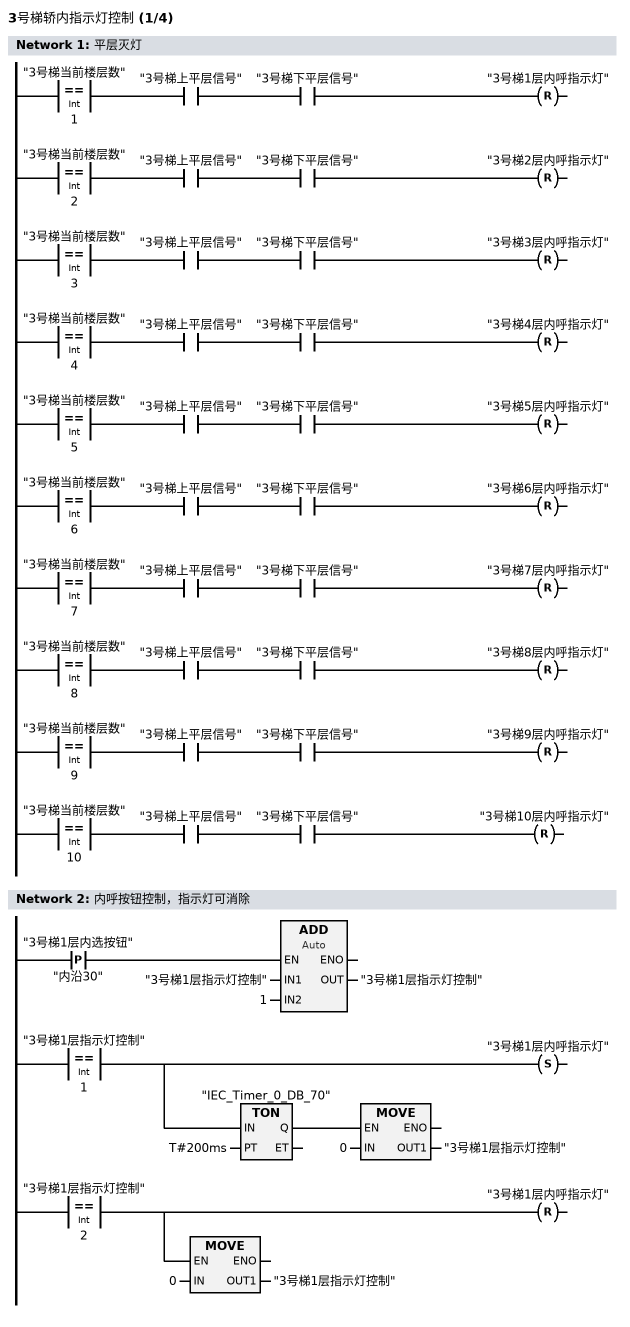
   RUNG wire#powerrail
      { S7_Templates := "SrcType := Int" } EQ_Contact(in1 := "3号梯当前楼层数", in2 := 1)
      Contact( "3号梯上平层信号" )
      Contact( "3号梯下平层信号" )
      R_Coil( "3号梯1层内呼指示灯" )
   END_RUNG
   RUNG wire#powerrail
      { S7_Templates := "SrcType := Int" } EQ_Contact(in1 := "3号梯当前楼层数", in2 := 2)
      Contact( "3号梯上平层信号" )
      Contact( "3号梯下平层信号" )
      R_Coil( "3号梯2层内呼指示灯" )
   END_RUNG
   RUNG wire#powerrail
      { S7_Templates := "SrcType := Int" } EQ_Contact(in1 := "3号梯当前楼层数", in2 := 3)
      Contact( "3号梯上平层信号" )
      Contact( "3号梯下平层信号" )
      R_Coil( "3号梯3层内呼指示灯" )
   END_RUNG
   RUNG wire#powerrail
      { S7_Templates := "SrcType := Int" } EQ_Contact(in1 := "3号梯当前楼层数", in2 := 4)
      Contact( "3号梯上平层信号" )
      Contact( "3号梯下平层信号" )
      R_Coil( "3号梯4层内呼指示灯" )
   END_RUNG
   RUNG wire#powerrail
      { S7_Templates := "SrcType := Int" } EQ_Contact(in1 := "3号梯当前楼层数", in2 := 5)
      Contact( "3号梯上平层信号" )
      Contact( "3号梯下平层信号" )
      R_Coil( "3号梯5层内呼指示灯" )
   END_RUNG
   RUNG wire#powerrail
      { S7_Templates := "SrcType := Int" } EQ_Contact(in1 := "3号梯当前楼层数", in2 := 6)
      Contact( "3号梯上平层信号" )
      Contact( "3号梯下平层信号" )
      R_Coil( "3号梯6层内呼指示灯" )
   END_RUNG
   RUNG wire#powerrail
      { S7_Templates := "SrcType := Int" } EQ_Contact(in1 := "3号梯当前楼层数", in2 := 7)
      Contact( "3号梯上平层信号" )
      Contact( "3号梯下平层信号" )
      R_Coil( "3号梯7层内呼指示灯" )
   END_RUNG
   RUNG wire#powerrail
      { S7_Templates := "SrcType := Int" } EQ_Contact(in1 := "3号梯当前楼层数", in2 := 8)
      Contact( "3号梯上平层信号" )
      Contact( "3号梯下平层信号" )
      R_Coil( "3号梯8层内呼指示灯" )
   END_RUNG
   RUNG wire#powerrail
      { S7_Templates := "SrcType := Int" } EQ_Contact(in1 := "3号梯当前楼层数", in2 := 9)
      Contact( "3号梯上平层信号" )
      Contact( "3号梯下平层信号" )
      R_Coil( "3号梯9层内呼指示灯" )
   END_RUNG
   RUNG wire#powerrail
      { S7_Templates := "SrcType := Int" } EQ_Contact(in1 := "3号梯当前楼层数", in2 := 10)
      Contact( "3号梯上平层信号" )
      Contact( "3号梯下平层信号" )
      R_Coil( "3号梯10层内呼指示灯" )
   END_RUNG
   // the same network as SCL:
   IF ("3号梯当前楼层数" = 1) AND "3号梯上平层信号" AND "3号梯下平层信号" THEN "3号梯1层内呼指示灯" := FALSE; END_IF;
   IF ("3号梯当前楼层数" = 2) AND "3号梯上平层信号" AND "3号梯下平层信号" THEN "3号梯2层内呼指示灯" := FALSE; END_IF;
   IF ("3号梯当前楼层数" = 3) AND "3号梯上平层信号" AND "3号梯下平层信号" THEN "3号梯3层内呼指示灯" := FALSE; END_IF;
   IF ("3号梯当前楼层数" = 4) AND "3号梯上平层信号" AND "3号梯下平层信号" THEN "3号梯4层内呼指示灯" := FALSE; END_IF;
   IF ("3号梯当前楼层数" = 5) AND "3号梯上平层信号" AND "3号梯下平层信号" THEN "3号梯5层内呼指示灯" := FALSE; END_IF;
   IF ("3号梯当前楼层数" = 6) AND "3号梯上平层信号" AND "3号梯下平层信号" THEN "3号梯6层内呼指示灯" := FALSE; END_IF;
   IF ("3号梯当前楼层数" = 7) AND "3号梯上平层信号" AND "3号梯下平层信号" THEN "3号梯7层内呼指示灯" := FALSE; END_IF;
   IF ("3号梯当前楼层数" = 8) AND "3号梯上平层信号" AND "3号梯下平层信号" THEN "3号梯8层内呼指示灯" := FALSE; END_IF;
   IF ("3号梯当前楼层数" = 9) AND "3号梯上平层信号" AND "3号梯下平层信号" THEN "3号梯9层内呼指示灯" := FALSE; END_IF;
   IF ("3号梯当前楼层数" = 10) AND "3号梯上平层信号" AND "3号梯下平层信号" THEN "3号梯10层内呼指示灯" := FALSE; END_IF;
END_REGION

REGION Network 2: 内呼按钮控制，指示灯可消除
   #_w1 := "3号梯1层内选按钮" AND NOT "内沿30";   // rising edge of "3号梯1层内选按钮"
   "内沿30" := "3号梯1层内选按钮";
   IF #_w1 THEN "3号梯1层指示灯控制" := "3号梯1层指示灯控制" + 1; END_IF;
   #_w2 := "3号梯1层指示灯控制" = 1;
   IF #_w2 THEN "3号梯1层内呼指示灯" := TRUE; END_IF;
   "IEC_Timer_0_DB_70".TON(IN := #_w2, PT := T#200ms);
   IF "IEC_Timer_0_DB_70".Q THEN "3号梯1层指示灯控制" := 0; END_IF;
   IF "3号梯1层指示灯控制" = 2 THEN
       "3号梯1层内呼指示灯" := FALSE;
       "3号梯1层指示灯控制" := 0;
   END_IF;
END_REGION

REGION Network 3: 内呼按钮控制，指示灯可消除
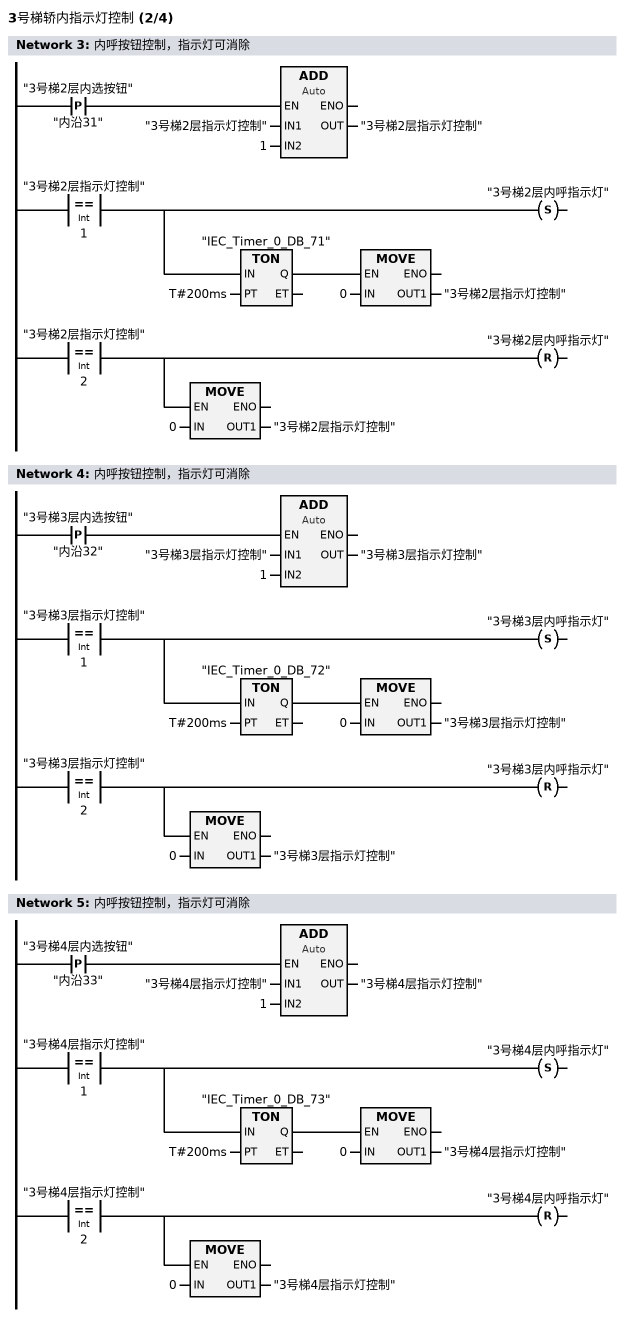
   #_w1 := "3号梯2层内选按钮" AND NOT "内沿31";   // rising edge of "3号梯2层内选按钮"
   "内沿31" := "3号梯2层内选按钮";
   IF #_w1 THEN "3号梯2层指示灯控制" := "3号梯2层指示灯控制" + 1; END_IF;
   #_w2 := "3号梯2层指示灯控制" = 1;
   IF #_w2 THEN "3号梯2层内呼指示灯" := TRUE; END_IF;
   "IEC_Timer_0_DB_71".TON(IN := #_w2, PT := T#200ms);
   IF "IEC_Timer_0_DB_71".Q THEN "3号梯2层指示灯控制" := 0; END_IF;
   IF "3号梯2层指示灯控制" = 2 THEN
       "3号梯2层内呼指示灯" := FALSE;
       "3号梯2层指示灯控制" := 0;
   END_IF;
END_REGION

REGION Network 4: 内呼按钮控制，指示灯可消除
   #_w1 := "3号梯3层内选按钮" AND NOT "内沿32";   // rising edge of "3号梯3层内选按钮"
   "内沿32" := "3号梯3层内选按钮";
   IF #_w1 THEN "3号梯3层指示灯控制" := "3号梯3层指示灯控制" + 1; END_IF;
   #_w2 := "3号梯3层指示灯控制" = 1;
   IF #_w2 THEN "3号梯3层内呼指示灯" := TRUE; END_IF;
   "IEC_Timer_0_DB_72".TON(IN := #_w2, PT := T#200ms);
   IF "IEC_Timer_0_DB_72".Q THEN "3号梯3层指示灯控制" := 0; END_IF;
   IF "3号梯3层指示灯控制" = 2 THEN
       "3号梯3层内呼指示灯" := FALSE;
       "3号梯3层指示灯控制" := 0;
   END_IF;
END_REGION

REGION Network 5: 内呼按钮控制，指示灯可消除
   #_w1 := "3号梯4层内选按钮" AND NOT "内沿33";   // rising edge of "3号梯4层内选按钮"
   "内沿33" := "3号梯4层内选按钮";
   IF #_w1 THEN "3号梯4层指示灯控制" := "3号梯4层指示灯控制" + 1; END_IF;
   #_w2 := "3号梯4层指示灯控制" = 1;
   IF #_w2 THEN "3号梯4层内呼指示灯" := TRUE; END_IF;
   "IEC_Timer_0_DB_73".TON(IN := #_w2, PT := T#200ms);
   IF "IEC_Timer_0_DB_73".Q THEN "3号梯4层指示灯控制" := 0; END_IF;
   IF "3号梯4层指示灯控制" = 2 THEN
       "3号梯4层内呼指示灯" := FALSE;
       "3号梯4层指示灯控制" := 0;
   END_IF;
END_REGION

REGION Network 6: 内呼按钮控制，指示灯可消除
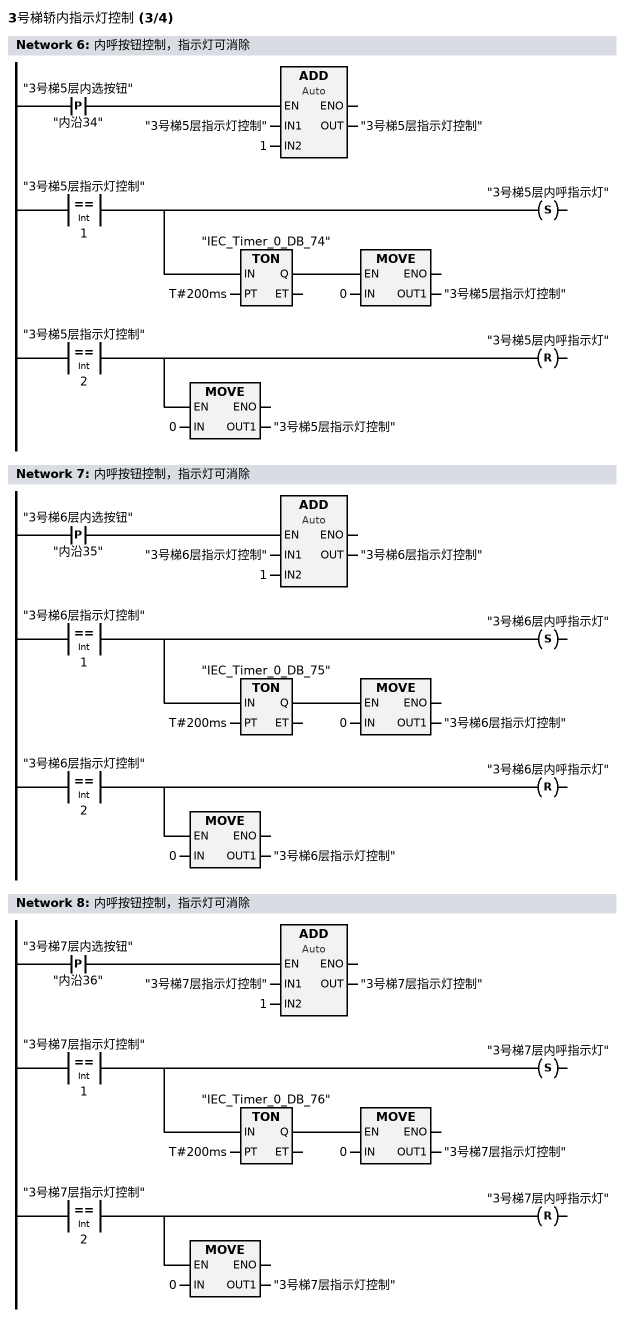
   #_w1 := "3号梯5层内选按钮" AND NOT "内沿34";   // rising edge of "3号梯5层内选按钮"
   "内沿34" := "3号梯5层内选按钮";
   IF #_w1 THEN "3号梯5层指示灯控制" := "3号梯5层指示灯控制" + 1; END_IF;
   #_w2 := "3号梯5层指示灯控制" = 1;
   IF #_w2 THEN "3号梯5层内呼指示灯" := TRUE; END_IF;
   "IEC_Timer_0_DB_74".TON(IN := #_w2, PT := T#200ms);
   IF "IEC_Timer_0_DB_74".Q THEN "3号梯5层指示灯控制" := 0; END_IF;
   IF "3号梯5层指示灯控制" = 2 THEN
       "3号梯5层内呼指示灯" := FALSE;
       "3号梯5层指示灯控制" := 0;
   END_IF;
END_REGION

REGION Network 7: 内呼按钮控制，指示灯可消除
   #_w1 := "3号梯6层内选按钮" AND NOT "内沿35";   // rising edge of "3号梯6层内选按钮"
   "内沿35" := "3号梯6层内选按钮";
   IF #_w1 THEN "3号梯6层指示灯控制" := "3号梯6层指示灯控制" + 1; END_IF;
   #_w2 := "3号梯6层指示灯控制" = 1;
   IF #_w2 THEN "3号梯6层内呼指示灯" := TRUE; END_IF;
   "IEC_Timer_0_DB_75".TON(IN := #_w2, PT := T#200ms);
   IF "IEC_Timer_0_DB_75".Q THEN "3号梯6层指示灯控制" := 0; END_IF;
   IF "3号梯6层指示灯控制" = 2 THEN
       "3号梯6层内呼指示灯" := FALSE;
       "3号梯6层指示灯控制" := 0;
   END_IF;
END_REGION

REGION Network 8: 内呼按钮控制，指示灯可消除
   #_w1 := "3号梯7层内选按钮" AND NOT "内沿36";   // rising edge of "3号梯7层内选按钮"
   "内沿36" := "3号梯7层内选按钮";
   IF #_w1 THEN "3号梯7层指示灯控制" := "3号梯7层指示灯控制" + 1; END_IF;
   #_w2 := "3号梯7层指示灯控制" = 1;
   IF #_w2 THEN "3号梯7层内呼指示灯" := TRUE; END_IF;
   "IEC_Timer_0_DB_76".TON(IN := #_w2, PT := T#200ms);
   IF "IEC_Timer_0_DB_76".Q THEN "3号梯7层指示灯控制" := 0; END_IF;
   IF "3号梯7层指示灯控制" = 2 THEN
       "3号梯7层内呼指示灯" := FALSE;
       "3号梯7层指示灯控制" := 0;
   END_IF;
END_REGION

REGION Network 9: 内呼按钮控制，指示灯可消除
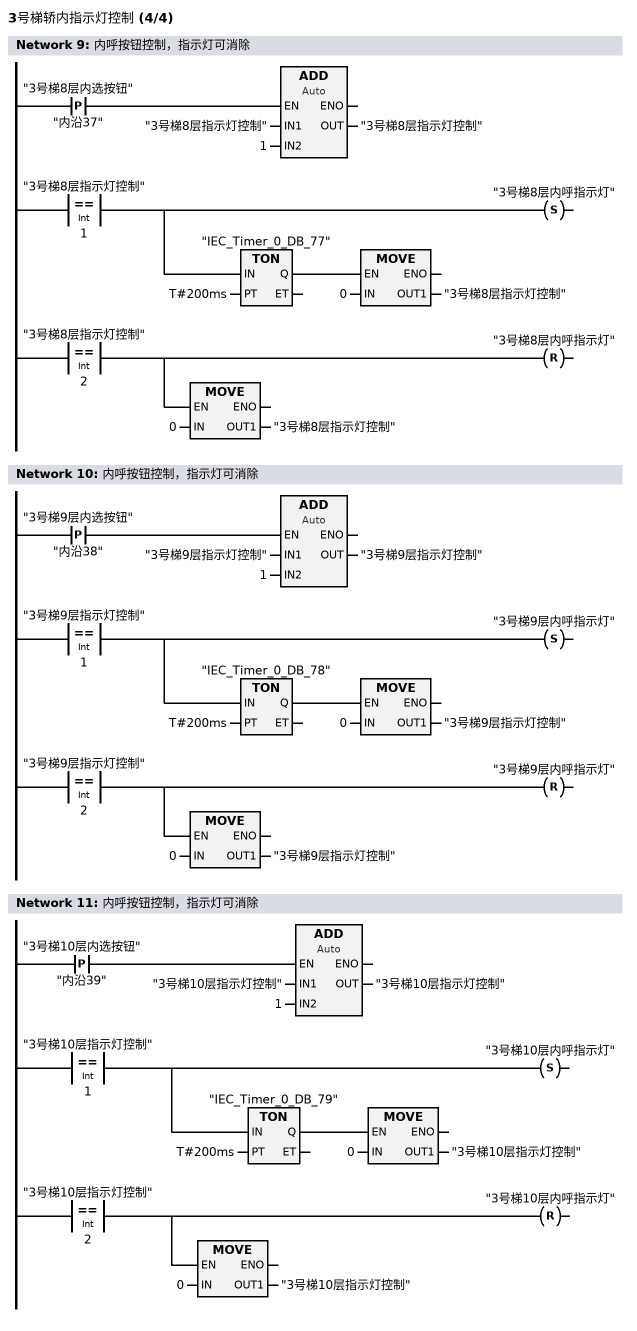
   #_w1 := "3号梯8层内选按钮" AND NOT "内沿37";   // rising edge of "3号梯8层内选按钮"
   "内沿37" := "3号梯8层内选按钮";
   IF #_w1 THEN "3号梯8层指示灯控制" := "3号梯8层指示灯控制" + 1; END_IF;
   #_w2 := "3号梯8层指示灯控制" = 1;
   IF #_w2 THEN "3号梯8层内呼指示灯" := TRUE; END_IF;
   "IEC_Timer_0_DB_77".TON(IN := #_w2, PT := T#200ms);
   IF "IEC_Timer_0_DB_77".Q THEN "3号梯8层指示灯控制" := 0; END_IF;
   IF "3号梯8层指示灯控制" = 2 THEN
       "3号梯8层内呼指示灯" := FALSE;
       "3号梯8层指示灯控制" := 0;
   END_IF;
END_REGION

REGION Network 10: 内呼按钮控制，指示灯可消除
   #_w1 := "3号梯9层内选按钮" AND NOT "内沿38";   // rising edge of "3号梯9层内选按钮"
   "内沿38" := "3号梯9层内选按钮";
   IF #_w1 THEN "3号梯9层指示灯控制" := "3号梯9层指示灯控制" + 1; END_IF;
   #_w2 := "3号梯9层指示灯控制" = 1;
   IF #_w2 THEN "3号梯9层内呼指示灯" := TRUE; END_IF;
   "IEC_Timer_0_DB_78".TON(IN := #_w2, PT := T#200ms);
   IF "IEC_Timer_0_DB_78".Q THEN "3号梯9层指示灯控制" := 0; END_IF;
   IF "3号梯9层指示灯控制" = 2 THEN
       "3号梯9层内呼指示灯" := FALSE;
       "3号梯9层指示灯控制" := 0;
   END_IF;
END_REGION

REGION Network 11: 内呼按钮控制，指示灯可消除
   #_w1 := "3号梯10层内选按钮" AND NOT "内沿39";   // rising edge of "3号梯10层内选按钮"
   "内沿39" := "3号梯10层内选按钮";
   IF #_w1 THEN "3号梯10层指示灯控制" := "3号梯10层指示灯控制" + 1; END_IF;
   #_w2 := "3号梯10层指示灯控制" = 1;
   IF #_w2 THEN "3号梯10层内呼指示灯" := TRUE; END_IF;
   "IEC_Timer_0_DB_79".TON(IN := #_w2, PT := T#200ms);
   IF "IEC_Timer_0_DB_79".Q THEN "3号梯10层指示灯控制" := 0; END_IF;
   IF "3号梯10层指示灯控制" = 2 THEN
       "3号梯10层内呼指示灯" := FALSE;
       "3号梯10层指示灯控制" := 0;
   END_IF;
END_REGION
END_FUNCTION

FUNCTION "3号梯保护程序" : Void   // FC41, LAD
{ S7_Optimized_Access := 'TRUE' }
VERSION : 0.1
BEGIN

REGION Network 1: 休眠管理
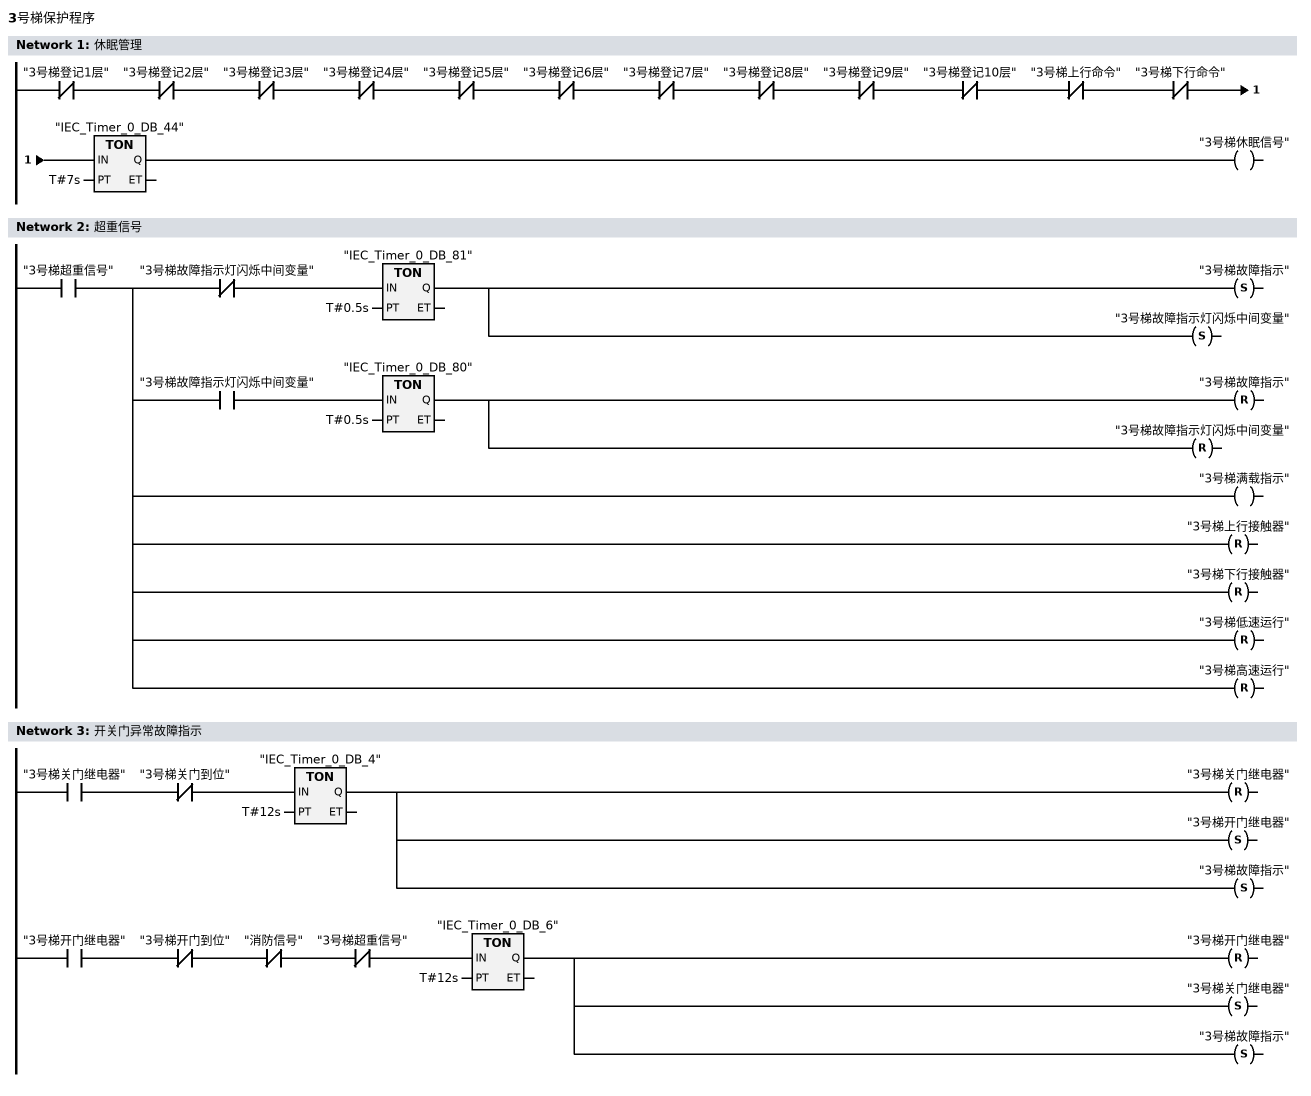
   "IEC_Timer_0_DB_44".TON(IN := NOT "3号梯登记1层" AND NOT "3号梯登记2层" AND NOT "3号梯登记3层" AND NOT "3号梯登记4层" AND NOT "3号梯登记5层" AND NOT "3号梯登记6层" AND NOT "3号梯登记7层" AND NOT "3号梯登记8层" AND NOT "3号梯登记9层" AND NOT "3号梯登记10层" AND NOT "3号梯上行命令" AND NOT "3号梯下行命令",
                           PT := T#7s);
   "3号梯休眠信号" := "IEC_Timer_0_DB_44".Q;
END_REGION

REGION Network 2: 超重信号
   "IEC_Timer_0_DB_81".TON(IN := "3号梯超重信号" AND NOT "3号梯故障指示灯闪烁中间变量", PT := T#0.5s);
   IF "IEC_Timer_0_DB_81".Q THEN
       "3号梯故障指示" := TRUE;
       "3号梯故障指示灯闪烁中间变量" := TRUE;
   END_IF;
   "IEC_Timer_0_DB_80".TON(IN := "3号梯超重信号" AND "3号梯故障指示灯闪烁中间变量", PT := T#0.5s);
   IF "IEC_Timer_0_DB_80".Q THEN
       "3号梯故障指示" := FALSE;
       "3号梯故障指示灯闪烁中间变量" := FALSE;
   END_IF;
   "3号梯满载指示" := "3号梯超重信号";
   IF "3号梯超重信号" THEN
       "3号梯上行接触器" := FALSE;
       "3号梯下行接触器" := FALSE;
       "3号梯低速运行" := FALSE;
       "3号梯高速运行" := FALSE;
   END_IF;
END_REGION

REGION Network 3: 开关门异常故障指示
   "IEC_Timer_0_DB_4".TON(IN := "3号梯关门继电器" AND NOT "3号梯关门到位", PT := T#12s);
   IF "IEC_Timer_0_DB_4".Q THEN
       "3号梯关门继电器" := FALSE;
       "3号梯开门继电器" := TRUE;
       "3号梯故障指示" := TRUE;
   END_IF;
   "IEC_Timer_0_DB_6".TON(IN := "3号梯开门继电器" AND NOT "3号梯开门到位" AND NOT "消防信号" AND NOT "3号梯超重信号", PT := T#12s);
   IF "IEC_Timer_0_DB_6".Q THEN
       "3号梯开门继电器" := FALSE;
       "3号梯关门继电器" := TRUE;
       "3号梯故障指示" := TRUE;
   END_IF;
END_REGION
END_FUNCTION

FUNCTION "2号梯保护程序" : Void   // FC42, LAD
{ S7_Optimized_Access := 'TRUE' }
VERSION : 0.1
BEGIN

REGION Network 1: 休眠管理
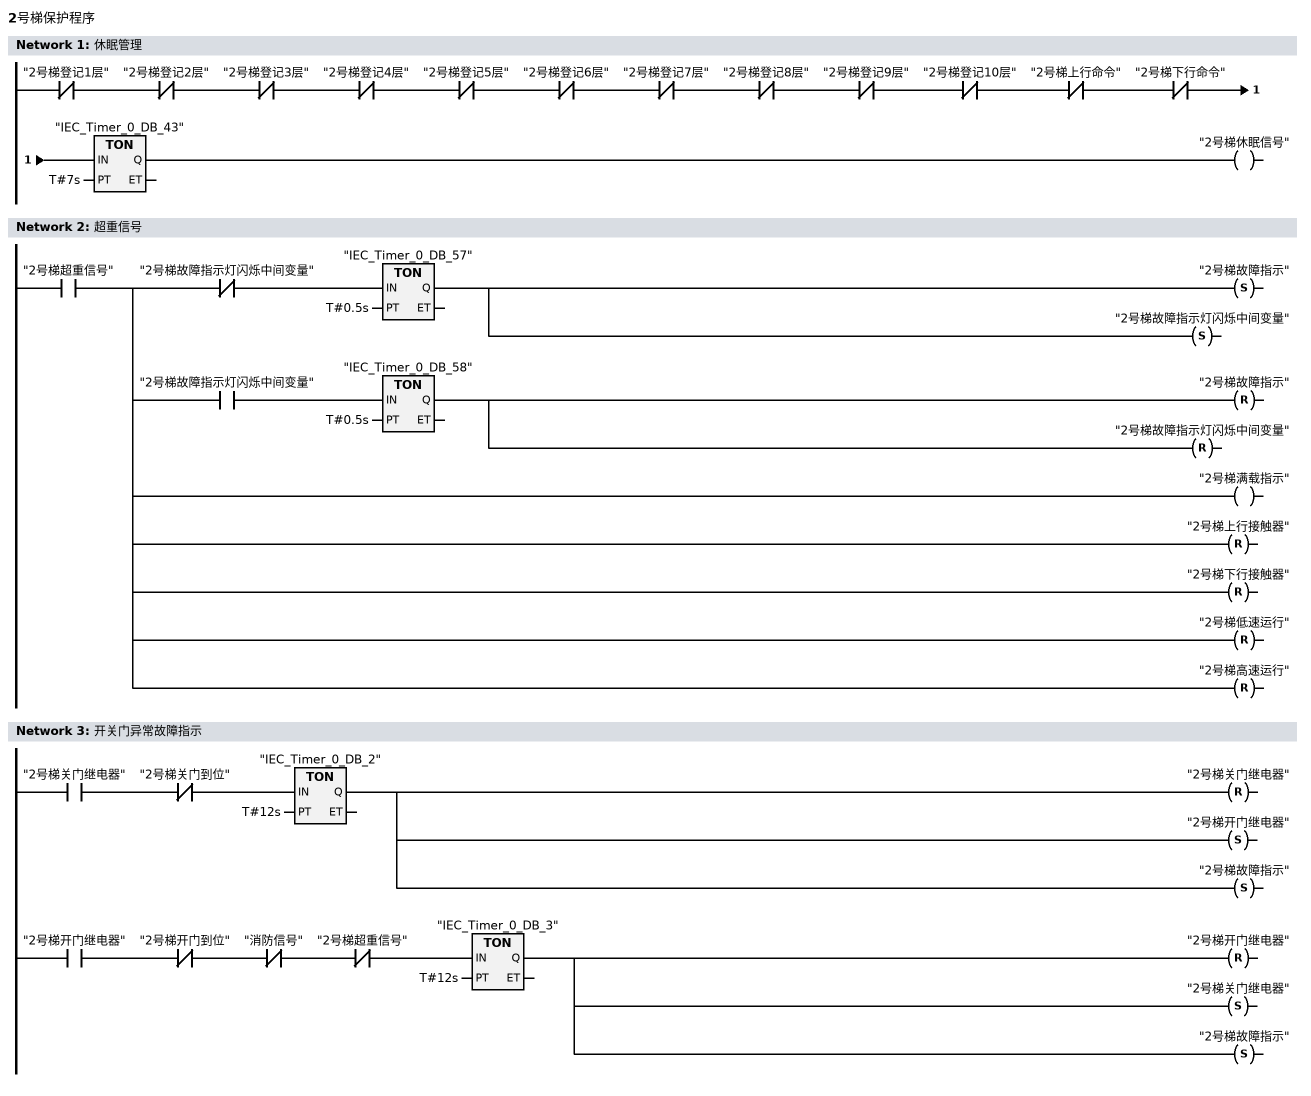
   "IEC_Timer_0_DB_43".TON(IN := NOT "2号梯登记1层" AND NOT "2号梯登记2层" AND NOT "2号梯登记3层" AND NOT "2号梯登记4层" AND NOT "2号梯登记5层" AND NOT "2号梯登记6层" AND NOT "2号梯登记7层" AND NOT "2号梯登记8层" AND NOT "2号梯登记9层" AND NOT "2号梯登记10层" AND NOT "2号梯上行命令" AND NOT "2号梯下行命令",
                           PT := T#7s);
   "2号梯休眠信号" := "IEC_Timer_0_DB_43".Q;
END_REGION

REGION Network 2: 超重信号
   "IEC_Timer_0_DB_57".TON(IN := "2号梯超重信号" AND NOT "2号梯故障指示灯闪烁中间变量", PT := T#0.5s);
   IF "IEC_Timer_0_DB_57".Q THEN
       "2号梯故障指示" := TRUE;
       "2号梯故障指示灯闪烁中间变量" := TRUE;
   END_IF;
   "IEC_Timer_0_DB_58".TON(IN := "2号梯超重信号" AND "2号梯故障指示灯闪烁中间变量", PT := T#0.5s);
   IF "IEC_Timer_0_DB_58".Q THEN
       "2号梯故障指示" := FALSE;
       "2号梯故障指示灯闪烁中间变量" := FALSE;
   END_IF;
   "2号梯满载指示" := "2号梯超重信号";
   IF "2号梯超重信号" THEN
       "2号梯上行接触器" := FALSE;
       "2号梯下行接触器" := FALSE;
       "2号梯低速运行" := FALSE;
       "2号梯高速运行" := FALSE;
   END_IF;
END_REGION

REGION Network 3: 开关门异常故障指示
   "IEC_Timer_0_DB_2".TON(IN := "2号梯关门继电器" AND NOT "2号梯关门到位", PT := T#12s);
   IF "IEC_Timer_0_DB_2".Q THEN
       "2号梯关门继电器" := FALSE;
       "2号梯开门继电器" := TRUE;
       "2号梯故障指示" := TRUE;
   END_IF;
   "IEC_Timer_0_DB_3".TON(IN := "2号梯开门继电器" AND NOT "2号梯开门到位" AND NOT "消防信号" AND NOT "2号梯超重信号", PT := T#12s);
   IF "IEC_Timer_0_DB_3".Q THEN
       "2号梯开门继电器" := FALSE;
       "2号梯关门继电器" := TRUE;
       "2号梯故障指示" := TRUE;
   END_IF;
END_REGION
END_FUNCTION

FUNCTION "3号梯错误指令消除" : Void   // FC43, LAD
{ S7_Optimized_Access := 'TRUE' }
VERSION : 0.1
BEGIN

REGION Network 1: 最上端/最下端时， 消除内呼信号
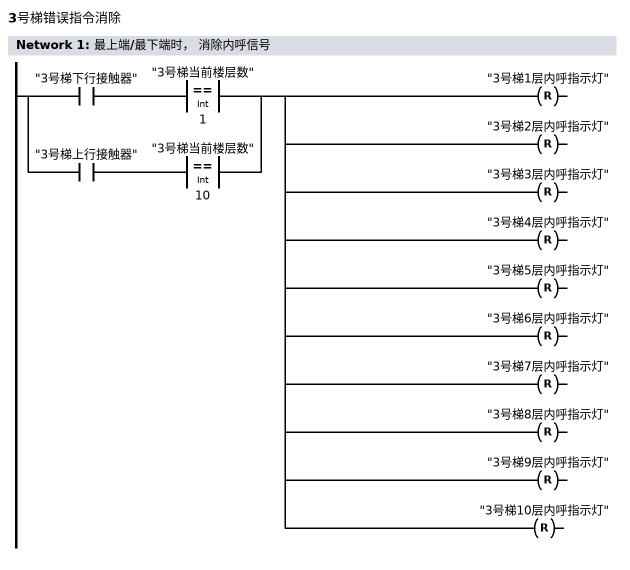
   RUNG wire#powerrail
      Contact( "3号梯下行接触器" )
      { S7_Templates := "SrcType := Int" } EQ_Contact(in1 := "3号梯当前楼层数", in2 := 1)
      wire#w1
      R_Coil( "3号梯1层内呼指示灯" )
   END_RUNG
   RUNG wire#powerrail
      Contact( "3号梯上行接触器" )
      { S7_Templates := "SrcType := Int" } EQ_Contact(in1 := "3号梯当前楼层数", in2 := 10)
   END_RUNG wire#w1
   RUNG wire#w1
      R_Coil( "3号梯2层内呼指示灯" )
   END_RUNG
   RUNG wire#w1
      R_Coil( "3号梯3层内呼指示灯" )
   END_RUNG
   RUNG wire#w1
      R_Coil( "3号梯4层内呼指示灯" )
   END_RUNG
   RUNG wire#w1
      R_Coil( "3号梯5层内呼指示灯" )
   END_RUNG
   RUNG wire#w1
      R_Coil( "3号梯6层内呼指示灯" )
   END_RUNG
   RUNG wire#w1
      R_Coil( "3号梯7层内呼指示灯" )
   END_RUNG
   RUNG wire#w1
      R_Coil( "3号梯8层内呼指示灯" )
   END_RUNG
   RUNG wire#w1
      R_Coil( "3号梯9层内呼指示灯" )
   END_RUNG
   RUNG wire#w1
      R_Coil( "3号梯10层内呼指示灯" )
   END_RUNG
   // the same network as SCL:
   IF ("3号梯下行接触器" AND ("3号梯当前楼层数" = 1)) OR ("3号梯上行接触器" AND ("3号梯当前楼层数" = 10)) THEN
       "3号梯1层内呼指示灯" := FALSE;
       "3号梯2层内呼指示灯" := FALSE;
       "3号梯3层内呼指示灯" := FALSE;
       "3号梯4层内呼指示灯" := FALSE;
       "3号梯5层内呼指示灯" := FALSE;
       "3号梯6层内呼指示灯" := FALSE;
       "3号梯7层内呼指示灯" := FALSE;
       "3号梯8层内呼指示灯" := FALSE;
       "3号梯9层内呼指示灯" := FALSE;
       "3号梯10层内呼指示灯" := FALSE;
   END_IF;
END_REGION
END_FUNCTION

FUNCTION "2号梯错误指令消除" : Void   // FC44, LAD
{ S7_Optimized_Access := 'TRUE' }
VERSION : 0.1
BEGIN

REGION Network 1: 最上端/最下端时， 消除内呼信号
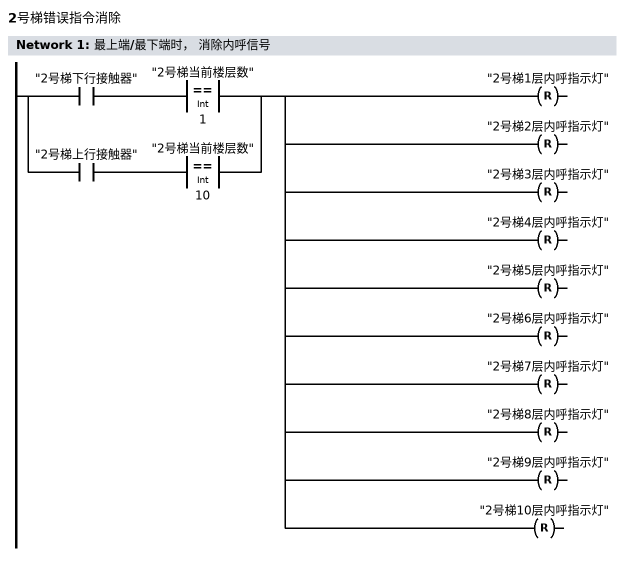
   RUNG wire#powerrail
      Contact( "2号梯下行接触器" )
      { S7_Templates := "SrcType := Int" } EQ_Contact(in1 := "2号梯当前楼层数", in2 := 1)
      wire#w1
      R_Coil( "2号梯1层内呼指示灯" )
   END_RUNG
   RUNG wire#powerrail
      Contact( "2号梯上行接触器" )
      { S7_Templates := "SrcType := Int" } EQ_Contact(in1 := "2号梯当前楼层数", in2 := 10)
   END_RUNG wire#w1
   RUNG wire#w1
      R_Coil( "2号梯2层内呼指示灯" )
   END_RUNG
   RUNG wire#w1
      R_Coil( "2号梯3层内呼指示灯" )
   END_RUNG
   RUNG wire#w1
      R_Coil( "2号梯4层内呼指示灯" )
   END_RUNG
   RUNG wire#w1
      R_Coil( "2号梯5层内呼指示灯" )
   END_RUNG
   RUNG wire#w1
      R_Coil( "2号梯6层内呼指示灯" )
   END_RUNG
   RUNG wire#w1
      R_Coil( "2号梯7层内呼指示灯" )
   END_RUNG
   RUNG wire#w1
      R_Coil( "2号梯8层内呼指示灯" )
   END_RUNG
   RUNG wire#w1
      R_Coil( "2号梯9层内呼指示灯" )
   END_RUNG
   RUNG wire#w1
      R_Coil( "2号梯10层内呼指示灯" )
   END_RUNG
   // the same network as SCL:
   IF ("2号梯下行接触器" AND ("2号梯当前楼层数" = 1)) OR ("2号梯上行接触器" AND ("2号梯当前楼层数" = 10)) THEN
       "2号梯1层内呼指示灯" := FALSE;
       "2号梯2层内呼指示灯" := FALSE;
       "2号梯3层内呼指示灯" := FALSE;
       "2号梯4层内呼指示灯" := FALSE;
       "2号梯5层内呼指示灯" := FALSE;
       "2号梯6层内呼指示灯" := FALSE;
       "2号梯7层内呼指示灯" := FALSE;
       "2号梯8层内呼指示灯" := FALSE;
       "2号梯9层内呼指示灯" := FALSE;
       "2号梯10层内呼指示灯" := FALSE;
   END_IF;
END_REGION
END_FUNCTION

FUNCTION "2号梯检修" : Void   // FC45, LAD
{ S7_Optimized_Access := 'TRUE' }
VERSION : 0.1
   VAR_TEMP   // added for the SCL form of the ladder/FBD networks
      _w1 : Bool;
   END_VAR
BEGIN

REGION Network 1: 检修
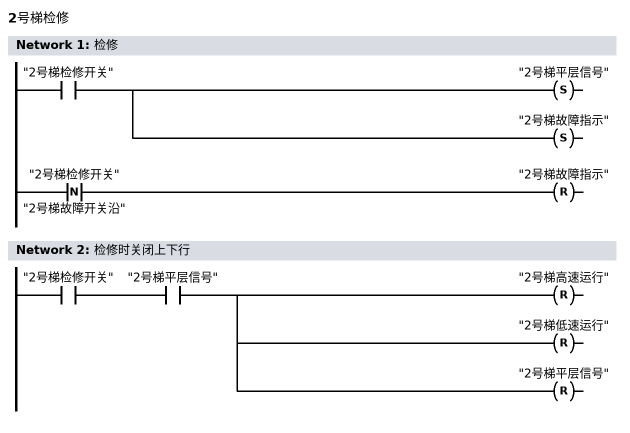
   RUNG wire#powerrail
      Contact( "2号梯检修开关" )
      wire#w1
      S_Coil( "2号梯平层信号" )
   END_RUNG
   RUNG wire#w1
      S_Coil( "2号梯故障指示" )
   END_RUNG
   RUNG wire#powerrail
      N_Contact(operand := "2号梯检修开关", bit := "2号梯故障开关沿")
      R_Coil( "2号梯故障指示" )
   END_RUNG
   // the same network as SCL:
   IF "2号梯检修开关" THEN
       "2号梯平层信号" := TRUE;
       "2号梯故障指示" := TRUE;
   END_IF;
   #_w1 := NOT "2号梯检修开关" AND "2号梯故障开关沿";   // falling edge of "2号梯检修开关"
   "2号梯故障开关沿" := "2号梯检修开关";
   IF #_w1 THEN "2号梯故障指示" := FALSE; END_IF;
END_REGION

REGION Network 2: 检修时关闭上下行
   RUNG wire#powerrail
      Contact( "2号梯检修开关" )
      Contact( "2号梯平层信号" )
      wire#w1
      R_Coil( "2号梯高速运行" )
   END_RUNG
   RUNG wire#w1
      R_Coil( "2号梯低速运行" )
   END_RUNG
   RUNG wire#w1
      R_Coil( "2号梯平层信号" )
   END_RUNG
   // the same network as SCL:
   IF "2号梯检修开关" AND "2号梯平层信号" THEN
       "2号梯高速运行" := FALSE;
       "2号梯低速运行" := FALSE;
       "2号梯平层信号" := FALSE;
   END_IF;
END_REGION
END_FUNCTION

FUNCTION "3号梯检修" : Void   // FC46, LAD
{ S7_Optimized_Access := 'TRUE' }
VERSION : 0.1
   VAR_TEMP   // added for the SCL form of the ladder/FBD networks
      _w1 : Bool;
   END_VAR
BEGIN

REGION Network 1: 检修
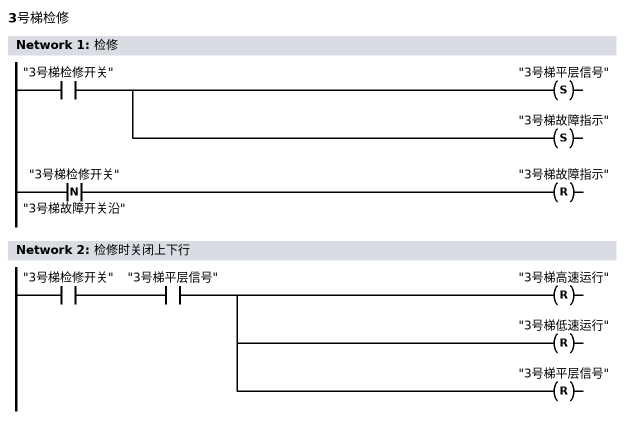
   RUNG wire#powerrail
      Contact( "3号梯检修开关" )
      wire#w1
      S_Coil( "3号梯平层信号" )
   END_RUNG
   RUNG wire#w1
      S_Coil( "3号梯故障指示" )
   END_RUNG
   RUNG wire#powerrail
      N_Contact(operand := "3号梯检修开关", bit := "3号梯故障开关沿")
      R_Coil( "3号梯故障指示" )
   END_RUNG
   // the same network as SCL:
   IF "3号梯检修开关" THEN
       "3号梯平层信号" := TRUE;
       "3号梯故障指示" := TRUE;
   END_IF;
   #_w1 := NOT "3号梯检修开关" AND "3号梯故障开关沿";   // falling edge of "3号梯检修开关"
   "3号梯故障开关沿" := "3号梯检修开关";
   IF #_w1 THEN "3号梯故障指示" := FALSE; END_IF;
END_REGION

REGION Network 2: 检修时关闭上下行
   RUNG wire#powerrail
      Contact( "3号梯检修开关" )
      Contact( "3号梯平层信号" )
      wire#w1
      R_Coil( "3号梯高速运行" )
   END_RUNG
   RUNG wire#w1
      R_Coil( "3号梯低速运行" )
   END_RUNG
   RUNG wire#w1
      R_Coil( "3号梯平层信号" )
   END_RUNG
   // the same network as SCL:
   IF "3号梯检修开关" AND "3号梯平层信号" THEN
       "3号梯高速运行" := FALSE;
       "3号梯低速运行" := FALSE;
       "3号梯平层信号" := FALSE;
   END_IF;
END_REGION
END_FUNCTION

FUNCTION "io_output" : Void   // FC47, LAD
{ S7_Optimized_Access := 'TRUE' }
VERSION : 0.1
BEGIN

REGION Network 1: 1号梯外呼上行绑定
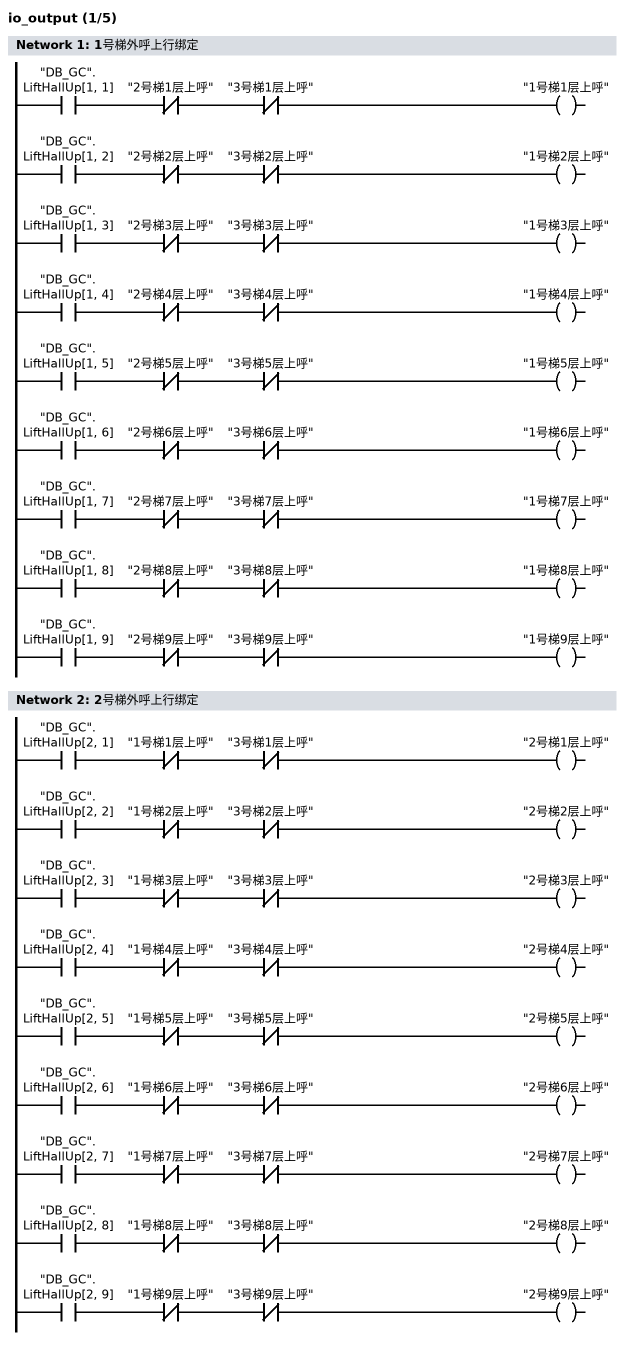
   RUNG wire#powerrail
      Contact( "DB_GC".LiftHallUp[1, 1] )
      I_Contact( "2号梯1层上呼" )
      I_Contact( "3号梯1层上呼" )
      Coil( "1号梯1层上呼" )
   END_RUNG
   RUNG wire#powerrail
      Contact( "DB_GC".LiftHallUp[1, 2] )
      I_Contact( "2号梯2层上呼" )
      I_Contact( "3号梯2层上呼" )
      Coil( "1号梯2层上呼" )
   END_RUNG
   RUNG wire#powerrail
      Contact( "DB_GC".LiftHallUp[1, 3] )
      I_Contact( "2号梯3层上呼" )
      I_Contact( "3号梯3层上呼" )
      Coil( "1号梯3层上呼" )
   END_RUNG
   RUNG wire#powerrail
      Contact( "DB_GC".LiftHallUp[1, 4] )
      I_Contact( "2号梯4层上呼" )
      I_Contact( "3号梯4层上呼" )
      Coil( "1号梯4层上呼" )
   END_RUNG
   RUNG wire#powerrail
      Contact( "DB_GC".LiftHallUp[1, 5] )
      I_Contact( "2号梯5层上呼" )
      I_Contact( "3号梯5层上呼" )
      Coil( "1号梯5层上呼" )
   END_RUNG
   RUNG wire#powerrail
      Contact( "DB_GC".LiftHallUp[1, 6] )
      I_Contact( "2号梯6层上呼" )
      I_Contact( "3号梯6层上呼" )
      Coil( "1号梯6层上呼" )
   END_RUNG
   RUNG wire#powerrail
      Contact( "DB_GC".LiftHallUp[1, 7] )
      I_Contact( "2号梯7层上呼" )
      I_Contact( "3号梯7层上呼" )
      Coil( "1号梯7层上呼" )
   END_RUNG
   RUNG wire#powerrail
      Contact( "DB_GC".LiftHallUp[1, 8] )
      I_Contact( "2号梯8层上呼" )
      I_Contact( "3号梯8层上呼" )
      Coil( "1号梯8层上呼" )
   END_RUNG
   RUNG wire#powerrail
      Contact( "DB_GC".LiftHallUp[1, 9] )
      I_Contact( "2号梯9层上呼" )
      I_Contact( "3号梯9层上呼" )
      Coil( "1号梯9层上呼" )
   END_RUNG
   // the same network as SCL:
   "1号梯1层上呼" := "DB_GC".LiftHallUp[1, 1] AND NOT "2号梯1层上呼" AND NOT "3号梯1层上呼";
   "1号梯2层上呼" := "DB_GC".LiftHallUp[1, 2] AND NOT "2号梯2层上呼" AND NOT "3号梯2层上呼";
   "1号梯3层上呼" := "DB_GC".LiftHallUp[1, 3] AND NOT "2号梯3层上呼" AND NOT "3号梯3层上呼";
   "1号梯4层上呼" := "DB_GC".LiftHallUp[1, 4] AND NOT "2号梯4层上呼" AND NOT "3号梯4层上呼";
   "1号梯5层上呼" := "DB_GC".LiftHallUp[1, 5] AND NOT "2号梯5层上呼" AND NOT "3号梯5层上呼";
   "1号梯6层上呼" := "DB_GC".LiftHallUp[1, 6] AND NOT "2号梯6层上呼" AND NOT "3号梯6层上呼";
   "1号梯7层上呼" := "DB_GC".LiftHallUp[1, 7] AND NOT "2号梯7层上呼" AND NOT "3号梯7层上呼";
   "1号梯8层上呼" := "DB_GC".LiftHallUp[1, 8] AND NOT "2号梯8层上呼" AND NOT "3号梯8层上呼";
   "1号梯9层上呼" := "DB_GC".LiftHallUp[1, 9] AND NOT "2号梯9层上呼" AND NOT "3号梯9层上呼";
END_REGION

REGION Network 2: 2号梯外呼上行绑定
   RUNG wire#powerrail
      Contact( "DB_GC".LiftHallUp[2, 1] )
      I_Contact( "1号梯1层上呼" )
      I_Contact( "3号梯1层上呼" )
      Coil( "2号梯1层上呼" )
   END_RUNG
   RUNG wire#powerrail
      Contact( "DB_GC".LiftHallUp[2, 2] )
      I_Contact( "1号梯2层上呼" )
      I_Contact( "3号梯2层上呼" )
      Coil( "2号梯2层上呼" )
   END_RUNG
   RUNG wire#powerrail
      Contact( "DB_GC".LiftHallUp[2, 3] )
      I_Contact( "1号梯3层上呼" )
      I_Contact( "3号梯3层上呼" )
      Coil( "2号梯3层上呼" )
   END_RUNG
   RUNG wire#powerrail
      Contact( "DB_GC".LiftHallUp[2, 4] )
      I_Contact( "1号梯4层上呼" )
      I_Contact( "3号梯4层上呼" )
      Coil( "2号梯4层上呼" )
   END_RUNG
   RUNG wire#powerrail
      Contact( "DB_GC".LiftHallUp[2, 5] )
      I_Contact( "1号梯5层上呼" )
      I_Contact( "3号梯5层上呼" )
      Coil( "2号梯5层上呼" )
   END_RUNG
   RUNG wire#powerrail
      Contact( "DB_GC".LiftHallUp[2, 6] )
      I_Contact( "1号梯6层上呼" )
      I_Contact( "3号梯6层上呼" )
      Coil( "2号梯6层上呼" )
   END_RUNG
   RUNG wire#powerrail
      Contact( "DB_GC".LiftHallUp[2, 7] )
      I_Contact( "1号梯7层上呼" )
      I_Contact( "3号梯7层上呼" )
      Coil( "2号梯7层上呼" )
   END_RUNG
   RUNG wire#powerrail
      Contact( "DB_GC".LiftHallUp[2, 8] )
      I_Contact( "1号梯8层上呼" )
      I_Contact( "3号梯8层上呼" )
      Coil( "2号梯8层上呼" )
   END_RUNG
   RUNG wire#powerrail
      Contact( "DB_GC".LiftHallUp[2, 9] )
      I_Contact( "1号梯9层上呼" )
      I_Contact( "3号梯9层上呼" )
      Coil( "2号梯9层上呼" )
   END_RUNG
   // the same network as SCL:
   "2号梯1层上呼" := "DB_GC".LiftHallUp[2, 1] AND NOT "1号梯1层上呼" AND NOT "3号梯1层上呼";
   "2号梯2层上呼" := "DB_GC".LiftHallUp[2, 2] AND NOT "1号梯2层上呼" AND NOT "3号梯2层上呼";
   "2号梯3层上呼" := "DB_GC".LiftHallUp[2, 3] AND NOT "1号梯3层上呼" AND NOT "3号梯3层上呼";
   "2号梯4层上呼" := "DB_GC".LiftHallUp[2, 4] AND NOT "1号梯4层上呼" AND NOT "3号梯4层上呼";
   "2号梯5层上呼" := "DB_GC".LiftHallUp[2, 5] AND NOT "1号梯5层上呼" AND NOT "3号梯5层上呼";
   "2号梯6层上呼" := "DB_GC".LiftHallUp[2, 6] AND NOT "1号梯6层上呼" AND NOT "3号梯6层上呼";
   "2号梯7层上呼" := "DB_GC".LiftHallUp[2, 7] AND NOT "1号梯7层上呼" AND NOT "3号梯7层上呼";
   "2号梯8层上呼" := "DB_GC".LiftHallUp[2, 8] AND NOT "1号梯8层上呼" AND NOT "3号梯8层上呼";
   "2号梯9层上呼" := "DB_GC".LiftHallUp[2, 9] AND NOT "1号梯9层上呼" AND NOT "3号梯9层上呼";
END_REGION

REGION Network 3: 3号梯外呼上行绑定
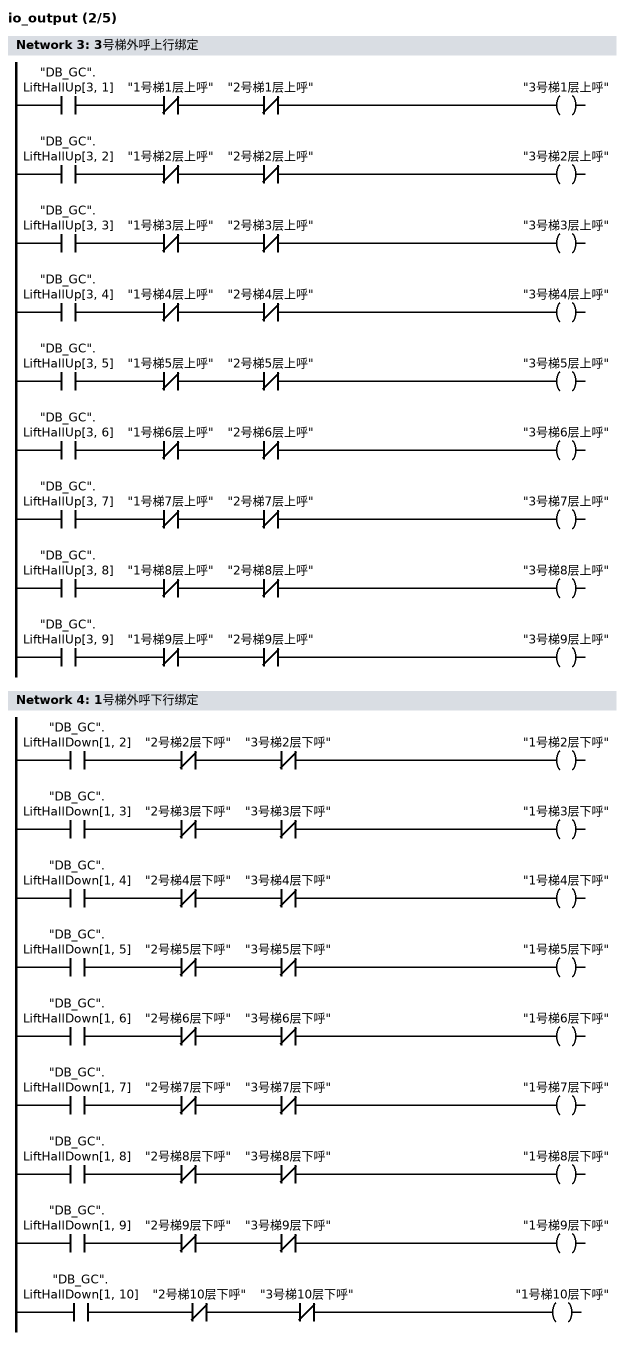
   RUNG wire#powerrail
      Contact( "DB_GC".LiftHallUp[3, 1] )
      I_Contact( "1号梯1层上呼" )
      I_Contact( "2号梯1层上呼" )
      Coil( "3号梯1层上呼" )
   END_RUNG
   RUNG wire#powerrail
      Contact( "DB_GC".LiftHallUp[3, 2] )
      I_Contact( "1号梯2层上呼" )
      I_Contact( "2号梯2层上呼" )
      Coil( "3号梯2层上呼" )
   END_RUNG
   RUNG wire#powerrail
      Contact( "DB_GC".LiftHallUp[3, 3] )
      I_Contact( "1号梯3层上呼" )
      I_Contact( "2号梯3层上呼" )
      Coil( "3号梯3层上呼" )
   END_RUNG
   RUNG wire#powerrail
      Contact( "DB_GC".LiftHallUp[3, 4] )
      I_Contact( "1号梯4层上呼" )
      I_Contact( "2号梯4层上呼" )
      Coil( "3号梯4层上呼" )
   END_RUNG
   RUNG wire#powerrail
      Contact( "DB_GC".LiftHallUp[3, 5] )
      I_Contact( "1号梯5层上呼" )
      I_Contact( "2号梯5层上呼" )
      Coil( "3号梯5层上呼" )
   END_RUNG
   RUNG wire#powerrail
      Contact( "DB_GC".LiftHallUp[3, 6] )
      I_Contact( "1号梯6层上呼" )
      I_Contact( "2号梯6层上呼" )
      Coil( "3号梯6层上呼" )
   END_RUNG
   RUNG wire#powerrail
      Contact( "DB_GC".LiftHallUp[3, 7] )
      I_Contact( "1号梯7层上呼" )
      I_Contact( "2号梯7层上呼" )
      Coil( "3号梯7层上呼" )
   END_RUNG
   RUNG wire#powerrail
      Contact( "DB_GC".LiftHallUp[3, 8] )
      I_Contact( "1号梯8层上呼" )
      I_Contact( "2号梯8层上呼" )
      Coil( "3号梯8层上呼" )
   END_RUNG
   RUNG wire#powerrail
      Contact( "DB_GC".LiftHallUp[3, 9] )
      I_Contact( "1号梯9层上呼" )
      I_Contact( "2号梯9层上呼" )
      Coil( "3号梯9层上呼" )
   END_RUNG
   // the same network as SCL:
   "3号梯1层上呼" := "DB_GC".LiftHallUp[3, 1] AND NOT "1号梯1层上呼" AND NOT "2号梯1层上呼";
   "3号梯2层上呼" := "DB_GC".LiftHallUp[3, 2] AND NOT "1号梯2层上呼" AND NOT "2号梯2层上呼";
   "3号梯3层上呼" := "DB_GC".LiftHallUp[3, 3] AND NOT "1号梯3层上呼" AND NOT "2号梯3层上呼";
   "3号梯4层上呼" := "DB_GC".LiftHallUp[3, 4] AND NOT "1号梯4层上呼" AND NOT "2号梯4层上呼";
   "3号梯5层上呼" := "DB_GC".LiftHallUp[3, 5] AND NOT "1号梯5层上呼" AND NOT "2号梯5层上呼";
   "3号梯6层上呼" := "DB_GC".LiftHallUp[3, 6] AND NOT "1号梯6层上呼" AND NOT "2号梯6层上呼";
   "3号梯7层上呼" := "DB_GC".LiftHallUp[3, 7] AND NOT "1号梯7层上呼" AND NOT "2号梯7层上呼";
   "3号梯8层上呼" := "DB_GC".LiftHallUp[3, 8] AND NOT "1号梯8层上呼" AND NOT "2号梯8层上呼";
   "3号梯9层上呼" := "DB_GC".LiftHallUp[3, 9] AND NOT "1号梯9层上呼" AND NOT "2号梯9层上呼";
END_REGION

REGION Network 4: 1号梯外呼下行绑定
   RUNG wire#powerrail
      Contact( "DB_GC".LiftHallDown[1, 2] )
      I_Contact( "2号梯2层下呼" )
      I_Contact( "3号梯2层下呼" )
      Coil( "1号梯2层下呼" )
   END_RUNG
   RUNG wire#powerrail
      Contact( "DB_GC".LiftHallDown[1, 3] )
      I_Contact( "2号梯3层下呼" )
      I_Contact( "3号梯3层下呼" )
      Coil( "1号梯3层下呼" )
   END_RUNG
   RUNG wire#powerrail
      Contact( "DB_GC".LiftHallDown[1, 4] )
      I_Contact( "2号梯4层下呼" )
      I_Contact( "3号梯4层下呼" )
      Coil( "1号梯4层下呼" )
   END_RUNG
   RUNG wire#powerrail
      Contact( "DB_GC".LiftHallDown[1, 5] )
      I_Contact( "2号梯5层下呼" )
      I_Contact( "3号梯5层下呼" )
      Coil( "1号梯5层下呼" )
   END_RUNG
   RUNG wire#powerrail
      Contact( "DB_GC".LiftHallDown[1, 6] )
      I_Contact( "2号梯6层下呼" )
      I_Contact( "3号梯6层下呼" )
      Coil( "1号梯6层下呼" )
   END_RUNG
   RUNG wire#powerrail
      Contact( "DB_GC".LiftHallDown[1, 7] )
      I_Contact( "2号梯7层下呼" )
      I_Contact( "3号梯7层下呼" )
      Coil( "1号梯7层下呼" )
   END_RUNG
   RUNG wire#powerrail
      Contact( "DB_GC".LiftHallDown[1, 8] )
      I_Contact( "2号梯8层下呼" )
      I_Contact( "3号梯8层下呼" )
      Coil( "1号梯8层下呼" )
   END_RUNG
   RUNG wire#powerrail
      Contact( "DB_GC".LiftHallDown[1, 9] )
      I_Contact( "2号梯9层下呼" )
      I_Contact( "3号梯9层下呼" )
      Coil( "1号梯9层下呼" )
   END_RUNG
   RUNG wire#powerrail
      Contact( "DB_GC".LiftHallDown[1, 10] )
      I_Contact( "2号梯10层下呼" )
      I_Contact( "3号梯10层下呼" )
      Coil( "1号梯10层下呼" )
   END_RUNG
   // the same network as SCL:
   "1号梯2层下呼" := "DB_GC".LiftHallDown[1, 2] AND NOT "2号梯2层下呼" AND NOT "3号梯2层下呼";
   "1号梯3层下呼" := "DB_GC".LiftHallDown[1, 3] AND NOT "2号梯3层下呼" AND NOT "3号梯3层下呼";
   "1号梯4层下呼" := "DB_GC".LiftHallDown[1, 4] AND NOT "2号梯4层下呼" AND NOT "3号梯4层下呼";
   "1号梯5层下呼" := "DB_GC".LiftHallDown[1, 5] AND NOT "2号梯5层下呼" AND NOT "3号梯5层下呼";
   "1号梯6层下呼" := "DB_GC".LiftHallDown[1, 6] AND NOT "2号梯6层下呼" AND NOT "3号梯6层下呼";
   "1号梯7层下呼" := "DB_GC".LiftHallDown[1, 7] AND NOT "2号梯7层下呼" AND NOT "3号梯7层下呼";
   "1号梯8层下呼" := "DB_GC".LiftHallDown[1, 8] AND NOT "2号梯8层下呼" AND NOT "3号梯8层下呼";
   "1号梯9层下呼" := "DB_GC".LiftHallDown[1, 9] AND NOT "2号梯9层下呼" AND NOT "3号梯9层下呼";
   "1号梯10层下呼" := "DB_GC".LiftHallDown[1, 10] AND NOT "2号梯10层下呼" AND NOT "3号梯10层下呼";
END_REGION

REGION Network 5: 2号梯外呼下行绑定
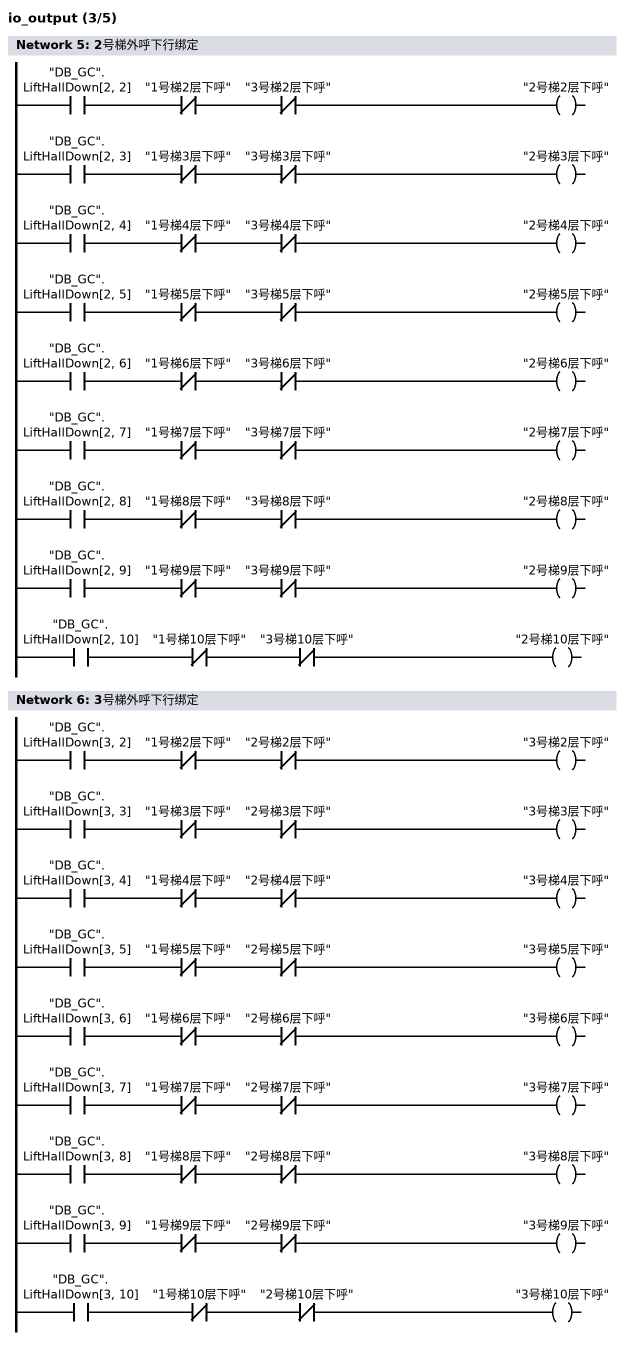
   RUNG wire#powerrail
      Contact( "DB_GC".LiftHallDown[2, 2] )
      I_Contact( "1号梯2层下呼" )
      I_Contact( "3号梯2层下呼" )
      Coil( "2号梯2层下呼" )
   END_RUNG
   RUNG wire#powerrail
      Contact( "DB_GC".LiftHallDown[2, 3] )
      I_Contact( "1号梯3层下呼" )
      I_Contact( "3号梯3层下呼" )
      Coil( "2号梯3层下呼" )
   END_RUNG
   RUNG wire#powerrail
      Contact( "DB_GC".LiftHallDown[2, 4] )
      I_Contact( "1号梯4层下呼" )
      I_Contact( "3号梯4层下呼" )
      Coil( "2号梯4层下呼" )
   END_RUNG
   RUNG wire#powerrail
      Contact( "DB_GC".LiftHallDown[2, 5] )
      I_Contact( "1号梯5层下呼" )
      I_Contact( "3号梯5层下呼" )
      Coil( "2号梯5层下呼" )
   END_RUNG
   RUNG wire#powerrail
      Contact( "DB_GC".LiftHallDown[2, 6] )
      I_Contact( "1号梯6层下呼" )
      I_Contact( "3号梯6层下呼" )
      Coil( "2号梯6层下呼" )
   END_RUNG
   RUNG wire#powerrail
      Contact( "DB_GC".LiftHallDown[2, 7] )
      I_Contact( "1号梯7层下呼" )
      I_Contact( "3号梯7层下呼" )
      Coil( "2号梯7层下呼" )
   END_RUNG
   RUNG wire#powerrail
      Contact( "DB_GC".LiftHallDown[2, 8] )
      I_Contact( "1号梯8层下呼" )
      I_Contact( "3号梯8层下呼" )
      Coil( "2号梯8层下呼" )
   END_RUNG
   RUNG wire#powerrail
      Contact( "DB_GC".LiftHallDown[2, 9] )
      I_Contact( "1号梯9层下呼" )
      I_Contact( "3号梯9层下呼" )
      Coil( "2号梯9层下呼" )
   END_RUNG
   RUNG wire#powerrail
      Contact( "DB_GC".LiftHallDown[2, 10] )
      I_Contact( "1号梯10层下呼" )
      I_Contact( "3号梯10层下呼" )
      Coil( "2号梯10层下呼" )
   END_RUNG
   // the same network as SCL:
   "2号梯2层下呼" := "DB_GC".LiftHallDown[2, 2] AND NOT "1号梯2层下呼" AND NOT "3号梯2层下呼";
   "2号梯3层下呼" := "DB_GC".LiftHallDown[2, 3] AND NOT "1号梯3层下呼" AND NOT "3号梯3层下呼";
   "2号梯4层下呼" := "DB_GC".LiftHallDown[2, 4] AND NOT "1号梯4层下呼" AND NOT "3号梯4层下呼";
   "2号梯5层下呼" := "DB_GC".LiftHallDown[2, 5] AND NOT "1号梯5层下呼" AND NOT "3号梯5层下呼";
   "2号梯6层下呼" := "DB_GC".LiftHallDown[2, 6] AND NOT "1号梯6层下呼" AND NOT "3号梯6层下呼";
   "2号梯7层下呼" := "DB_GC".LiftHallDown[2, 7] AND NOT "1号梯7层下呼" AND NOT "3号梯7层下呼";
   "2号梯8层下呼" := "DB_GC".LiftHallDown[2, 8] AND NOT "1号梯8层下呼" AND NOT "3号梯8层下呼";
   "2号梯9层下呼" := "DB_GC".LiftHallDown[2, 9] AND NOT "1号梯9层下呼" AND NOT "3号梯9层下呼";
   "2号梯10层下呼" := "DB_GC".LiftHallDown[2, 10] AND NOT "1号梯10层下呼" AND NOT "3号梯10层下呼";
END_REGION

REGION Network 6: 3号梯外呼下行绑定
   RUNG wire#powerrail
      Contact( "DB_GC".LiftHallDown[3, 2] )
      I_Contact( "1号梯2层下呼" )
      I_Contact( "2号梯2层下呼" )
      Coil( "3号梯2层下呼" )
   END_RUNG
   RUNG wire#powerrail
      Contact( "DB_GC".LiftHallDown[3, 3] )
      I_Contact( "1号梯3层下呼" )
      I_Contact( "2号梯3层下呼" )
      Coil( "3号梯3层下呼" )
   END_RUNG
   RUNG wire#powerrail
      Contact( "DB_GC".LiftHallDown[3, 4] )
      I_Contact( "1号梯4层下呼" )
      I_Contact( "2号梯4层下呼" )
      Coil( "3号梯4层下呼" )
   END_RUNG
   RUNG wire#powerrail
      Contact( "DB_GC".LiftHallDown[3, 5] )
      I_Contact( "1号梯5层下呼" )
      I_Contact( "2号梯5层下呼" )
      Coil( "3号梯5层下呼" )
   END_RUNG
   RUNG wire#powerrail
      Contact( "DB_GC".LiftHallDown[3, 6] )
      I_Contact( "1号梯6层下呼" )
      I_Contact( "2号梯6层下呼" )
      Coil( "3号梯6层下呼" )
   END_RUNG
   RUNG wire#powerrail
      Contact( "DB_GC".LiftHallDown[3, 7] )
      I_Contact( "1号梯7层下呼" )
      I_Contact( "2号梯7层下呼" )
      Coil( "3号梯7层下呼" )
   END_RUNG
   RUNG wire#powerrail
      Contact( "DB_GC".LiftHallDown[3, 8] )
      I_Contact( "1号梯8层下呼" )
      I_Contact( "2号梯8层下呼" )
      Coil( "3号梯8层下呼" )
   END_RUNG
   RUNG wire#powerrail
      Contact( "DB_GC".LiftHallDown[3, 9] )
      I_Contact( "1号梯9层下呼" )
      I_Contact( "2号梯9层下呼" )
      Coil( "3号梯9层下呼" )
   END_RUNG
   RUNG wire#powerrail
      Contact( "DB_GC".LiftHallDown[3, 10] )
      I_Contact( "1号梯10层下呼" )
      I_Contact( "2号梯10层下呼" )
      Coil( "3号梯10层下呼" )
   END_RUNG
   // the same network as SCL:
   "3号梯2层下呼" := "DB_GC".LiftHallDown[3, 2] AND NOT "1号梯2层下呼" AND NOT "2号梯2层下呼";
   "3号梯3层下呼" := "DB_GC".LiftHallDown[3, 3] AND NOT "1号梯3层下呼" AND NOT "2号梯3层下呼";
   "3号梯4层下呼" := "DB_GC".LiftHallDown[3, 4] AND NOT "1号梯4层下呼" AND NOT "2号梯4层下呼";
   "3号梯5层下呼" := "DB_GC".LiftHallDown[3, 5] AND NOT "1号梯5层下呼" AND NOT "2号梯5层下呼";
   "3号梯6层下呼" := "DB_GC".LiftHallDown[3, 6] AND NOT "1号梯6层下呼" AND NOT "2号梯6层下呼";
   "3号梯7层下呼" := "DB_GC".LiftHallDown[3, 7] AND NOT "1号梯7层下呼" AND NOT "2号梯7层下呼";
   "3号梯8层下呼" := "DB_GC".LiftHallDown[3, 8] AND NOT "1号梯8层下呼" AND NOT "2号梯8层下呼";
   "3号梯9层下呼" := "DB_GC".LiftHallDown[3, 9] AND NOT "1号梯9层下呼" AND NOT "2号梯9层下呼";
   "3号梯10层下呼" := "DB_GC".LiftHallDown[3, 10] AND NOT "1号梯10层下呼" AND NOT "2号梯10层下呼";
END_REGION

REGION Network 7: 外呼上行指示灯灭灯
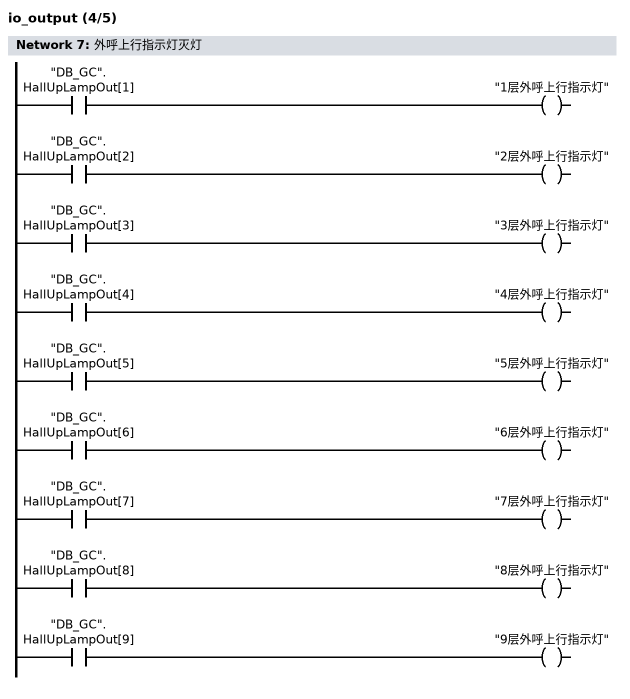
   RUNG wire#powerrail
      Contact( "DB_GC".HallUpLampOut[1] )
      Coil( "1层外呼上行指示灯" )
   END_RUNG
   RUNG wire#powerrail
      Contact( "DB_GC".HallUpLampOut[2] )
      Coil( "2层外呼上行指示灯" )
   END_RUNG
   RUNG wire#powerrail
      Contact( "DB_GC".HallUpLampOut[3] )
      Coil( "3层外呼上行指示灯" )
   END_RUNG
   RUNG wire#powerrail
      Contact( "DB_GC".HallUpLampOut[4] )
      Coil( "4层外呼上行指示灯" )
   END_RUNG
   RUNG wire#powerrail
      Contact( "DB_GC".HallUpLampOut[5] )
      Coil( "5层外呼上行指示灯" )
   END_RUNG
   RUNG wire#powerrail
      Contact( "DB_GC".HallUpLampOut[6] )
      Coil( "6层外呼上行指示灯" )
   END_RUNG
   RUNG wire#powerrail
      Contact( "DB_GC".HallUpLampOut[7] )
      Coil( "7层外呼上行指示灯" )
   END_RUNG
   RUNG wire#powerrail
      Contact( "DB_GC".HallUpLampOut[8] )
      Coil( "8层外呼上行指示灯" )
   END_RUNG
   RUNG wire#powerrail
      Contact( "DB_GC".HallUpLampOut[9] )
      Coil( "9层外呼上行指示灯" )
   END_RUNG
   // the same network as SCL:
   "1层外呼上行指示灯" := "DB_GC".HallUpLampOut[1];
   "2层外呼上行指示灯" := "DB_GC".HallUpLampOut[2];
   "3层外呼上行指示灯" := "DB_GC".HallUpLampOut[3];
   "4层外呼上行指示灯" := "DB_GC".HallUpLampOut[4];
   "5层外呼上行指示灯" := "DB_GC".HallUpLampOut[5];
   "6层外呼上行指示灯" := "DB_GC".HallUpLampOut[6];
   "7层外呼上行指示灯" := "DB_GC".HallUpLampOut[7];
   "8层外呼上行指示灯" := "DB_GC".HallUpLampOut[8];
   "9层外呼上行指示灯" := "DB_GC".HallUpLampOut[9];
END_REGION

REGION Network 8: 外呼上行指示灯灭灯
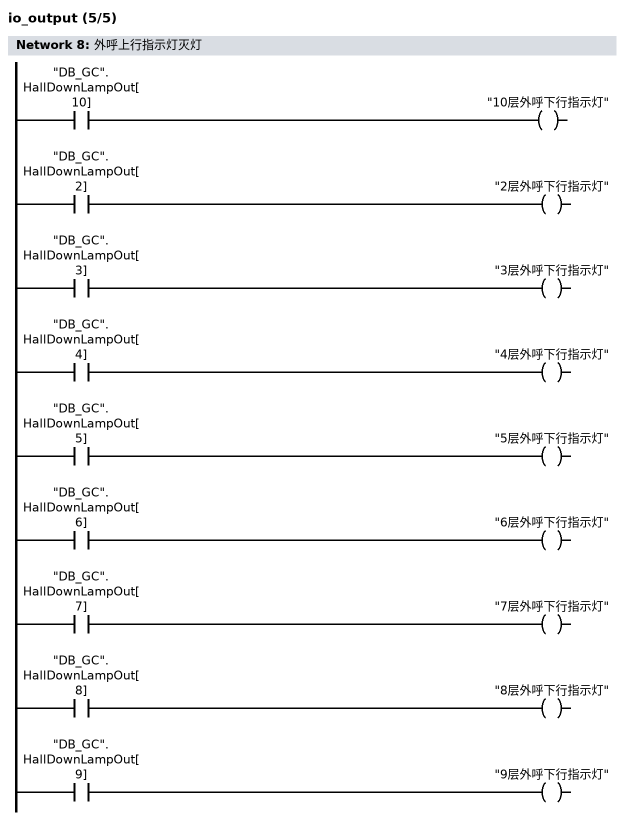
   RUNG wire#powerrail
      Contact( "DB_GC".HallDownLampOut[10] )
      Coil( "10层外呼下行指示灯" )
   END_RUNG
   RUNG wire#powerrail
      Contact( "DB_GC".HallDownLampOut[2] )
      Coil( "2层外呼下行指示灯" )
   END_RUNG
   RUNG wire#powerrail
      Contact( "DB_GC".HallDownLampOut[3] )
      Coil( "3层外呼下行指示灯" )
   END_RUNG
   RUNG wire#powerrail
      Contact( "DB_GC".HallDownLampOut[4] )
      Coil( "4层外呼下行指示灯" )
   END_RUNG
   RUNG wire#powerrail
      Contact( "DB_GC".HallDownLampOut[5] )
      Coil( "5层外呼下行指示灯" )
   END_RUNG
   RUNG wire#powerrail
      Contact( "DB_GC".HallDownLampOut[6] )
      Coil( "6层外呼下行指示灯" )
   END_RUNG
   RUNG wire#powerrail
      Contact( "DB_GC".HallDownLampOut[7] )
      Coil( "7层外呼下行指示灯" )
   END_RUNG
   RUNG wire#powerrail
      Contact( "DB_GC".HallDownLampOut[8] )
      Coil( "8层外呼下行指示灯" )
   END_RUNG
   RUNG wire#powerrail
      Contact( "DB_GC".HallDownLampOut[9] )
      Coil( "9层外呼下行指示灯" )
   END_RUNG
   // the same network as SCL:
   "10层外呼下行指示灯" := "DB_GC".HallDownLampOut[10];
   "2层外呼下行指示灯" := "DB_GC".HallDownLampOut[2];
   "3层外呼下行指示灯" := "DB_GC".HallDownLampOut[3];
   "4层外呼下行指示灯" := "DB_GC".HallDownLampOut[4];
   "5层外呼下行指示灯" := "DB_GC".HallDownLampOut[5];
   "6层外呼下行指示灯" := "DB_GC".HallDownLampOut[6];
   "7层外呼下行指示灯" := "DB_GC".HallDownLampOut[7];
   "8层外呼下行指示灯" := "DB_GC".HallDownLampOut[8];
   "9层外呼下行指示灯" := "DB_GC".HallDownLampOut[9];
END_REGION
END_FUNCTION

FUNCTION "3号梯开关门控制" : Void   // FC48, LAD
{ S7_Optimized_Access := 'TRUE' }
VERSION : 0.1
   VAR_TEMP   // added for the SCL form of the ladder/FBD networks
      _w1 : Bool;
   END_VAR
BEGIN

REGION Network 1: 开门使能
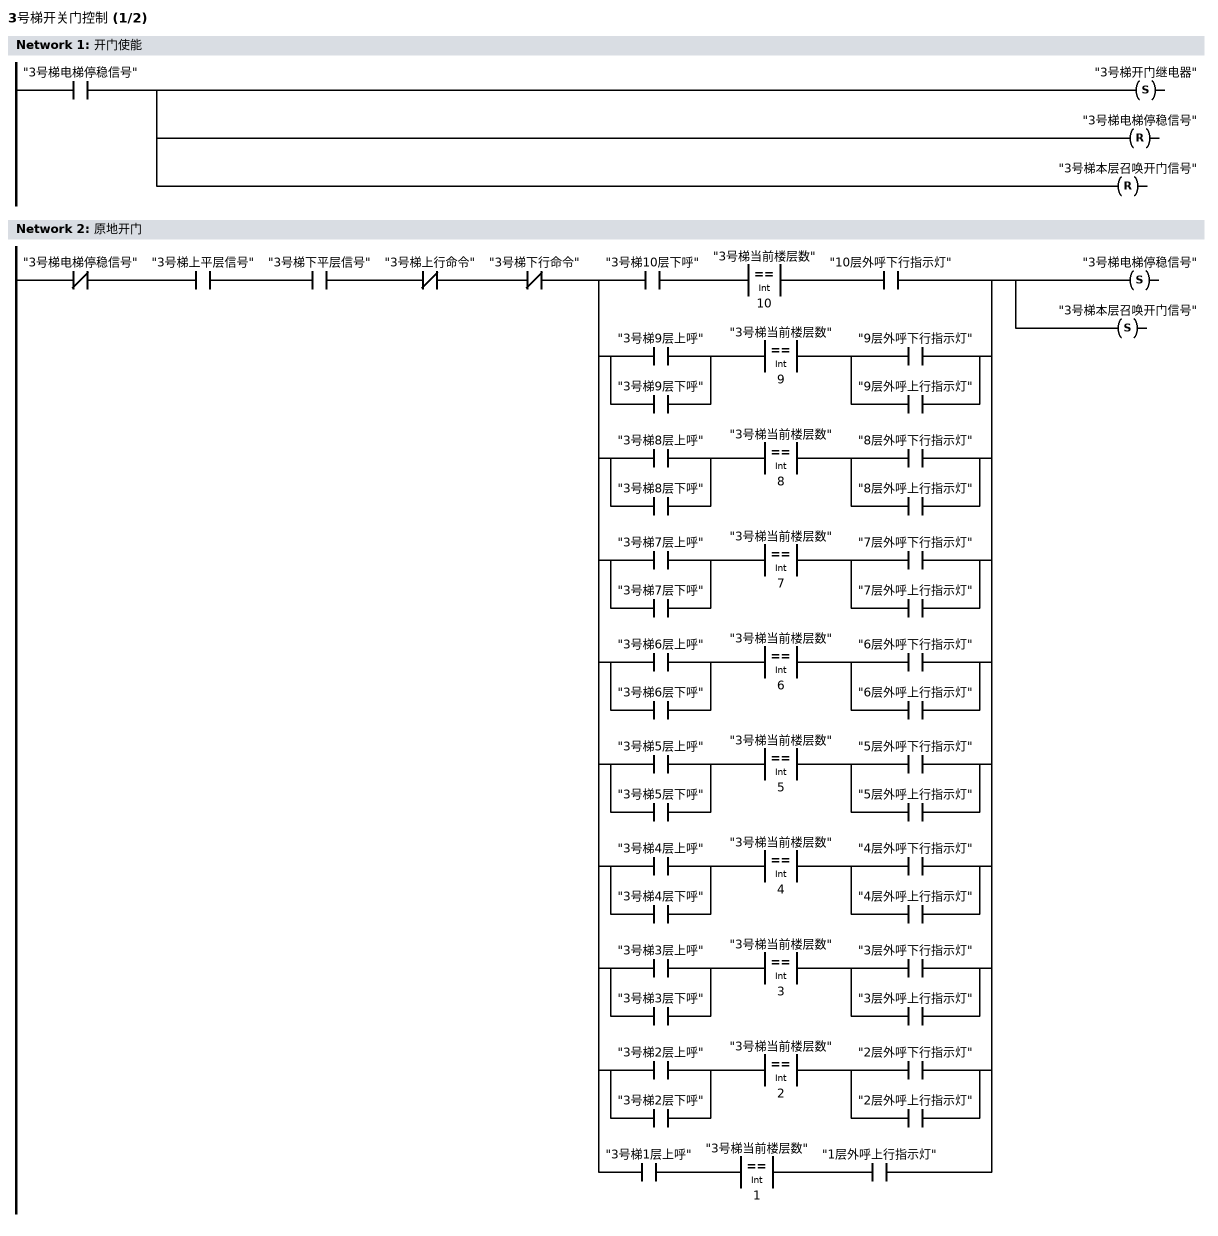
   RUNG wire#powerrail
      Contact( "3号梯电梯停稳信号" )
      wire#w1
      S_Coil( "3号梯开门继电器" )
   END_RUNG
   RUNG wire#w1
      R_Coil( "3号梯电梯停稳信号" )
   END_RUNG
   RUNG wire#w1
      R_Coil( "3号梯本层召唤开门信号" )
   END_RUNG
   // the same network as SCL:
   IF "3号梯电梯停稳信号" THEN "3号梯开门继电器" := TRUE; END_IF;
   #_w1 := "3号梯电梯停稳信号";
   IF #_w1 THEN
       "3号梯电梯停稳信号" := FALSE;
       "3号梯本层召唤开门信号" := FALSE;
   END_IF;
END_REGION

REGION Network 2: 原地开门
   RUNG wire#powerrail
      I_Contact( "3号梯电梯停稳信号" )
      Contact( "3号梯上平层信号" )
      Contact( "3号梯下平层信号" )
      I_Contact( "3号梯上行命令" )
      I_Contact( "3号梯下行命令" )
      wire#w1
      Contact( "3号梯10层下呼" )
      { S7_Templates := "SrcType := Int" } EQ_Contact(in1 := "3号梯当前楼层数", in2 := 10)
      Contact( "10层外呼下行指示灯" )
      wire#w2
      S_Coil( "3号梯电梯停稳信号" )
   END_RUNG
   RUNG wire#w1
      Contact( "3号梯9层上呼" )
      wire#w3
      { S7_Templates := "SrcType := Int" } EQ_Contact(in1 := "3号梯当前楼层数", in2 := 9)
      wire#w4
      Contact( "9层外呼下行指示灯" )
   END_RUNG wire#w2
   RUNG wire#w1
      Contact( "3号梯9层下呼" )
   END_RUNG wire#w3
   RUNG wire#w4
      Contact( "9层外呼上行指示灯" )
   END_RUNG wire#w2
   RUNG wire#w1
      Contact( "3号梯8层上呼" )
      wire#w5
      { S7_Templates := "SrcType := Int" } EQ_Contact(in1 := "3号梯当前楼层数", in2 := 8)
      wire#w6
      Contact( "8层外呼下行指示灯" )
   END_RUNG wire#w2
   RUNG wire#w1
      Contact( "3号梯8层下呼" )
   END_RUNG wire#w5
   RUNG wire#w6
      Contact( "8层外呼上行指示灯" )
   END_RUNG wire#w2
   RUNG wire#w1
      Contact( "3号梯7层上呼" )
      wire#w7
      { S7_Templates := "SrcType := Int" } EQ_Contact(in1 := "3号梯当前楼层数", in2 := 7)
      wire#w8
      Contact( "7层外呼下行指示灯" )
   END_RUNG wire#w2
   RUNG wire#w1
      Contact( "3号梯7层下呼" )
   END_RUNG wire#w7
   RUNG wire#w8
      Contact( "7层外呼上行指示灯" )
   END_RUNG wire#w2
   RUNG wire#w1
      Contact( "3号梯6层上呼" )
      wire#w9
      { S7_Templates := "SrcType := Int" } EQ_Contact(in1 := "3号梯当前楼层数", in2 := 6)
      wire#w10
      Contact( "6层外呼下行指示灯" )
   END_RUNG wire#w2
   RUNG wire#w1
      Contact( "3号梯6层下呼" )
   END_RUNG wire#w9
   RUNG wire#w10
      Contact( "6层外呼上行指示灯" )
   END_RUNG wire#w2
   RUNG wire#w1
      Contact( "3号梯5层上呼" )
      wire#w11
      { S7_Templates := "SrcType := Int" } EQ_Contact(in1 := "3号梯当前楼层数", in2 := 5)
      wire#w12
      Contact( "5层外呼下行指示灯" )
   END_RUNG wire#w2
   RUNG wire#w1
      Contact( "3号梯5层下呼" )
   END_RUNG wire#w11
   RUNG wire#w12
      Contact( "5层外呼上行指示灯" )
   END_RUNG wire#w2
   RUNG wire#w1
      Contact( "3号梯4层上呼" )
      wire#w13
      { S7_Templates := "SrcType := Int" } EQ_Contact(in1 := "3号梯当前楼层数", in2 := 4)
      wire#w14
      Contact( "4层外呼下行指示灯" )
   END_RUNG wire#w2
   RUNG wire#w1
      Contact( "3号梯4层下呼" )
   END_RUNG wire#w13
   RUNG wire#w14
      Contact( "4层外呼上行指示灯" )
   END_RUNG wire#w2
   RUNG wire#w1
      Contact( "3号梯3层上呼" )
      wire#w15
      { S7_Templates := "SrcType := Int" } EQ_Contact(in1 := "3号梯当前楼层数", in2 := 3)
      wire#w16
      Contact( "3层外呼下行指示灯" )
   END_RUNG wire#w2
   RUNG wire#w1
      Contact( "3号梯3层下呼" )
   END_RUNG wire#w15
   RUNG wire#w16
      Contact( "3层外呼上行指示灯" )
   END_RUNG wire#w2
   RUNG wire#w1
      Contact( "3号梯2层上呼" )
      wire#w17
      { S7_Templates := "SrcType := Int" } EQ_Contact(in1 := "3号梯当前楼层数", in2 := 2)
      wire#w18
      Contact( "2层外呼下行指示灯" )
   END_RUNG wire#w2
   RUNG wire#w1
      Contact( "3号梯2层下呼" )
   END_RUNG wire#w17
   RUNG wire#w18
      Contact( "2层外呼上行指示灯" )
   END_RUNG wire#w2
   RUNG wire#w1
      Contact( "3号梯1层上呼" )
      { S7_Templates := "SrcType := Int" } EQ_Contact(in1 := "3号梯当前楼层数", in2 := 1)
      Contact( "1层外呼上行指示灯" )
   END_RUNG wire#w2
   RUNG wire#w2
      S_Coil( "3号梯本层召唤开门信号" )
   END_RUNG
   // the same network as SCL:
   #_w1 := NOT "3号梯电梯停稳信号" AND "3号梯上平层信号" AND "3号梯下平层信号" AND NOT "3号梯上行命令" AND NOT "3号梯下行命令" AND (("3号梯10层下呼" AND ("3号梯当前楼层数" = 10) AND "10层外呼下行指示灯") OR (("3号梯9层上呼" OR "3号梯9层下呼") AND ("3号梯当前楼层数" = 9) AND ("9层外呼下行指示灯" OR "9层外呼上行指示灯")) OR (("3号梯8层上呼" OR "3号梯8层下呼") AND ("3号梯当前楼层数" = 8) AND ("8层外呼下行指示灯" OR "8层外呼上行指示灯")) OR (("3号梯7层上呼" OR "3号梯7层下呼") AND ("3号梯当前楼层数" = 7) AND ("7层外呼下行指示灯" OR "7层外呼上行指示灯")) OR (("3号梯6层上呼" OR "3号梯6层下呼") AND ("3号梯当前楼层数" = 6) AND ("6层外呼下行指示灯" OR "6层外呼上行指示灯")) OR (("3号梯5层上呼" OR "3号梯5层下呼") AND ("3号梯当前楼层数" = 5) AND ("5层外呼下行指示灯" OR "5层外呼上行指示灯")) OR (("3号梯4层上呼" OR "3号梯4层下呼") AND ("3号梯当前楼层数" = 4) AND ("4层外呼下行指示灯" OR "4层外呼上行指示灯")) OR (("3号梯3层上呼" OR "3号梯3层下呼") AND ("3号梯当前楼层数" = 3) AND ("3层外呼下行指示灯" OR "3层外呼上行指示灯")) OR (("3号梯2层上呼" OR "3号梯2层下呼") AND ("3号梯当前楼层数" = 2) AND ("2层外呼下行指示灯" OR "2层外呼上行指示灯")) OR ("3号梯1层上呼" AND ("3号梯当前楼层数" = 1) AND "1层外呼上行指示灯"));
   IF #_w1 THEN
       "3号梯电梯停稳信号" := TRUE;
       "3号梯本层召唤开门信号" := TRUE;
   END_IF;
END_REGION

REGION Network 3: 关门
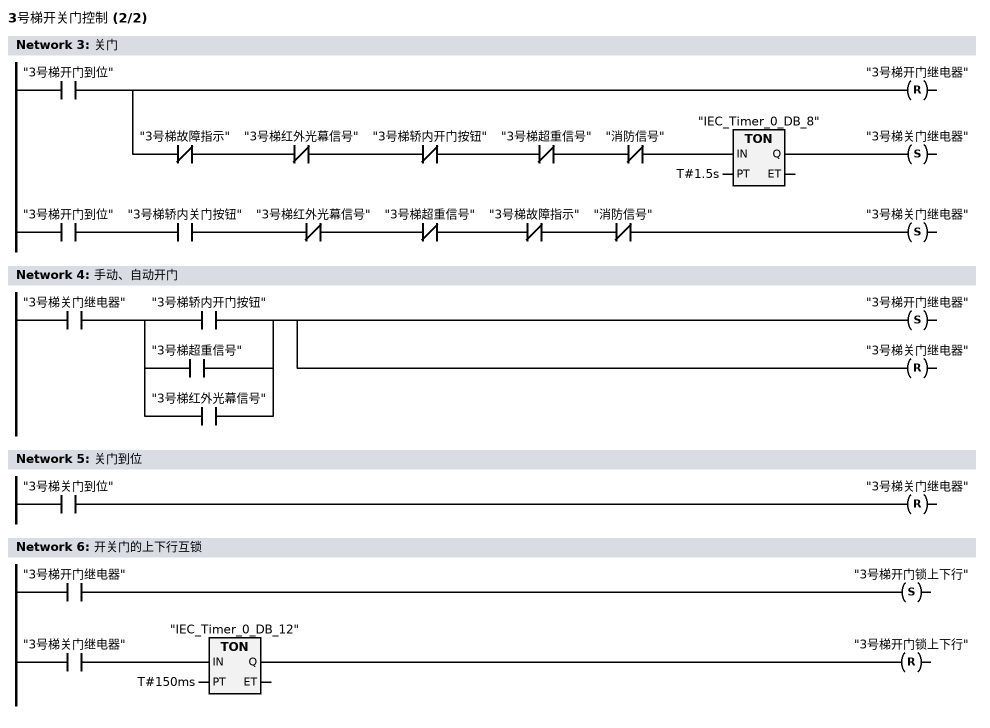
   IF "3号梯开门到位" THEN "3号梯开门继电器" := FALSE; END_IF;
   "IEC_Timer_0_DB_8".TON(IN := "3号梯开门到位" AND NOT "3号梯故障指示" AND NOT "3号梯红外光幕信号" AND NOT "3号梯轿内开门按钮" AND NOT "3号梯超重信号" AND NOT "消防信号",
                          PT := T#1.5s);
   IF "IEC_Timer_0_DB_8".Q THEN "3号梯关门继电器" := TRUE; END_IF;
   IF "3号梯开门到位" AND "3号梯轿内关门按钮" AND NOT "3号梯红外光幕信号" AND NOT "3号梯超重信号" AND NOT "3号梯故障指示" AND NOT "消防信号" THEN
       "3号梯关门继电器" := TRUE;
   END_IF;
END_REGION

REGION Network 4: 手动、自动开门
   RUNG wire#powerrail
      Contact( "3号梯关门继电器" )
      wire#w1
      Contact( "3号梯轿内开门按钮" )
      wire#w2
      S_Coil( "3号梯开门继电器" )
   END_RUNG
   RUNG wire#w1
      Contact( "3号梯超重信号" )
   END_RUNG wire#w2
   RUNG wire#w1
      Contact( "3号梯红外光幕信号" )
   END_RUNG wire#w2
   RUNG wire#w2
      R_Coil( "3号梯关门继电器" )
   END_RUNG
   // the same network as SCL:
   IF "3号梯关门继电器" AND ("3号梯轿内开门按钮" OR "3号梯超重信号" OR "3号梯红外光幕信号") THEN
       "3号梯开门继电器" := TRUE;
       "3号梯关门继电器" := FALSE;
   END_IF;
END_REGION

REGION Network 5: 关门到位
   RUNG wire#powerrail
      Contact( "3号梯关门到位" )
      R_Coil( "3号梯关门继电器" )
   END_RUNG
   // the same network as SCL:
   IF "3号梯关门到位" THEN "3号梯关门继电器" := FALSE; END_IF;
END_REGION

REGION Network 6: 开关门的上下行互锁
   IF "3号梯开门继电器" THEN "3号梯开门锁上下行" := TRUE; END_IF;
   "IEC_Timer_0_DB_12".TON(IN := "3号梯关门继电器", PT := T#150ms);
   IF "IEC_Timer_0_DB_12".Q THEN "3号梯开门锁上下行" := FALSE; END_IF;
END_REGION
END_FUNCTION

ORGANIZATION_BLOCK "Main"   // OB1, LAD, ProgramCycle
TITLE = "Main Program Sweep (Cycle)"
{ S7_Optimized_Access := 'TRUE' }
VERSION : 0.1
   VAR_INPUT
      Initial_Call : Bool;   // Initial call of this OB
      Remanence : Bool;   // =True, if remanent data are available
   END_VAR
BEGIN

REGION Network 1: 准备就绪延时
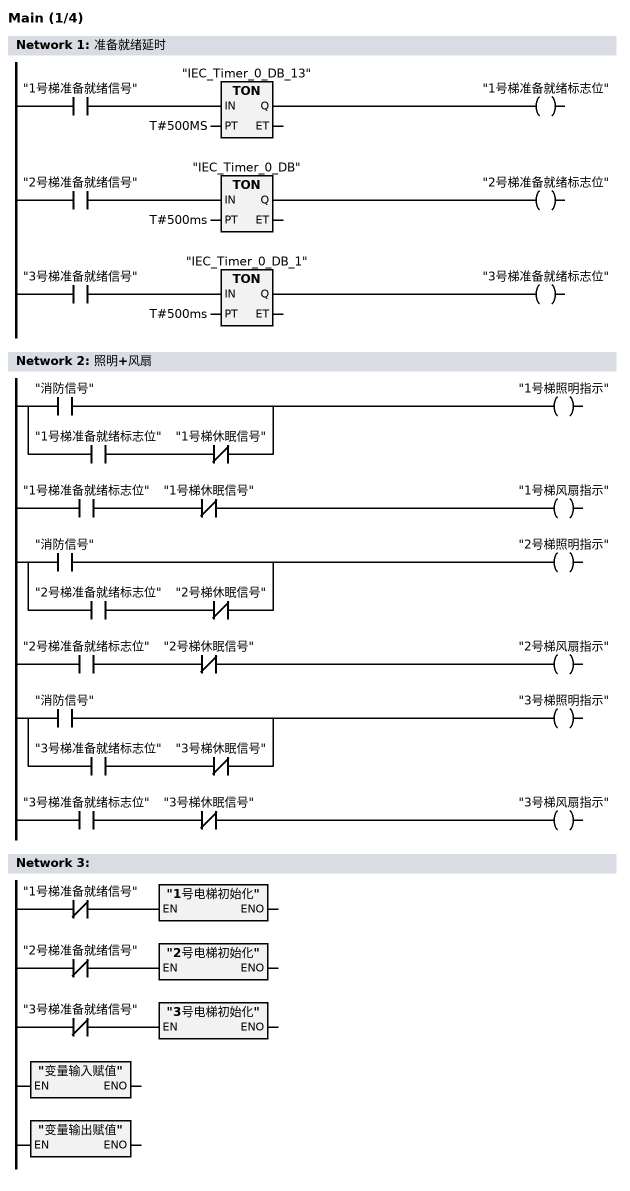
   "IEC_Timer_0_DB_13".TON(IN := "1号梯准备就绪信号", PT := T#500MS);
   "1号梯准备就绪标志位" := "IEC_Timer_0_DB_13".Q;
   "IEC_Timer_0_DB".TON(IN := "2号梯准备就绪信号", PT := T#500ms);
   "2号梯准备就绪标志位" := "IEC_Timer_0_DB".Q;
   "IEC_Timer_0_DB_1".TON(IN := "3号梯准备就绪信号", PT := T#500ms);
   "3号梯准备就绪标志位" := "IEC_Timer_0_DB_1".Q;
END_REGION

REGION Network 2: 照明+风扇
   RUNG wire#powerrail
      Contact( "消防信号" )
      wire#w1
      Coil( "1号梯照明指示" )
   END_RUNG
   RUNG wire#powerrail
      Contact( "1号梯准备就绪标志位" )
      I_Contact( "1号梯休眠信号" )
   END_RUNG wire#w1
   RUNG wire#powerrail
      Contact( "1号梯准备就绪标志位" )
      I_Contact( "1号梯休眠信号" )
      Coil( "1号梯风扇指示" )
   END_RUNG
   RUNG wire#powerrail
      Contact( "消防信号" )
      wire#w2
      Coil( "2号梯照明指示" )
   END_RUNG
   RUNG wire#powerrail
      Contact( "2号梯准备就绪标志位" )
      I_Contact( "2号梯休眠信号" )
   END_RUNG wire#w2
   RUNG wire#powerrail
      Contact( "2号梯准备就绪标志位" )
      I_Contact( "2号梯休眠信号" )
      Coil( "2号梯风扇指示" )
   END_RUNG
   RUNG wire#powerrail
      Contact( "消防信号" )
      wire#w3
      Coil( "3号梯照明指示" )
   END_RUNG
   RUNG wire#powerrail
      Contact( "3号梯准备就绪标志位" )
      I_Contact( "3号梯休眠信号" )
   END_RUNG wire#w3
   RUNG wire#powerrail
      Contact( "3号梯准备就绪标志位" )
      I_Contact( "3号梯休眠信号" )
      Coil( "3号梯风扇指示" )
   END_RUNG
   // the same network as SCL:
   "1号梯照明指示" := "消防信号" OR ("1号梯准备就绪标志位" AND NOT "1号梯休眠信号");
   "1号梯风扇指示" := "1号梯准备就绪标志位" AND NOT "1号梯休眠信号";
   "2号梯照明指示" := "消防信号" OR ("2号梯准备就绪标志位" AND NOT "2号梯休眠信号");
   "2号梯风扇指示" := "2号梯准备就绪标志位" AND NOT "2号梯休眠信号";
   "3号梯照明指示" := "消防信号" OR ("3号梯准备就绪标志位" AND NOT "3号梯休眠信号");
   "3号梯风扇指示" := "3号梯准备就绪标志位" AND NOT "3号梯休眠信号";
END_REGION

REGION Network 3
   RUNG wire#powerrail
      I_Contact( "1号梯准备就绪信号" )
      "1号电梯初始化"()
   END_RUNG
   RUNG wire#powerrail
      I_Contact( "2号梯准备就绪信号" )
      "2号电梯初始化"()
   END_RUNG
   RUNG wire#powerrail
      I_Contact( "3号梯准备就绪信号" )
      "3号电梯初始化"()
   END_RUNG
   RUNG wire#powerrail
      "变量输入赋值"()
   END_RUNG
   RUNG wire#powerrail
      "变量输出赋值"()
   END_RUNG
   // the same network as SCL:
   IF NOT "1号梯准备就绪信号" THEN "1号电梯初始化"(); END_IF;
   IF NOT "2号梯准备就绪信号" THEN "2号电梯初始化"(); END_IF;
   IF NOT "3号梯准备就绪信号" THEN "3号电梯初始化"(); END_IF;
   "变量输入赋值"();
   "变量输出赋值"();
END_REGION

REGION Network 4
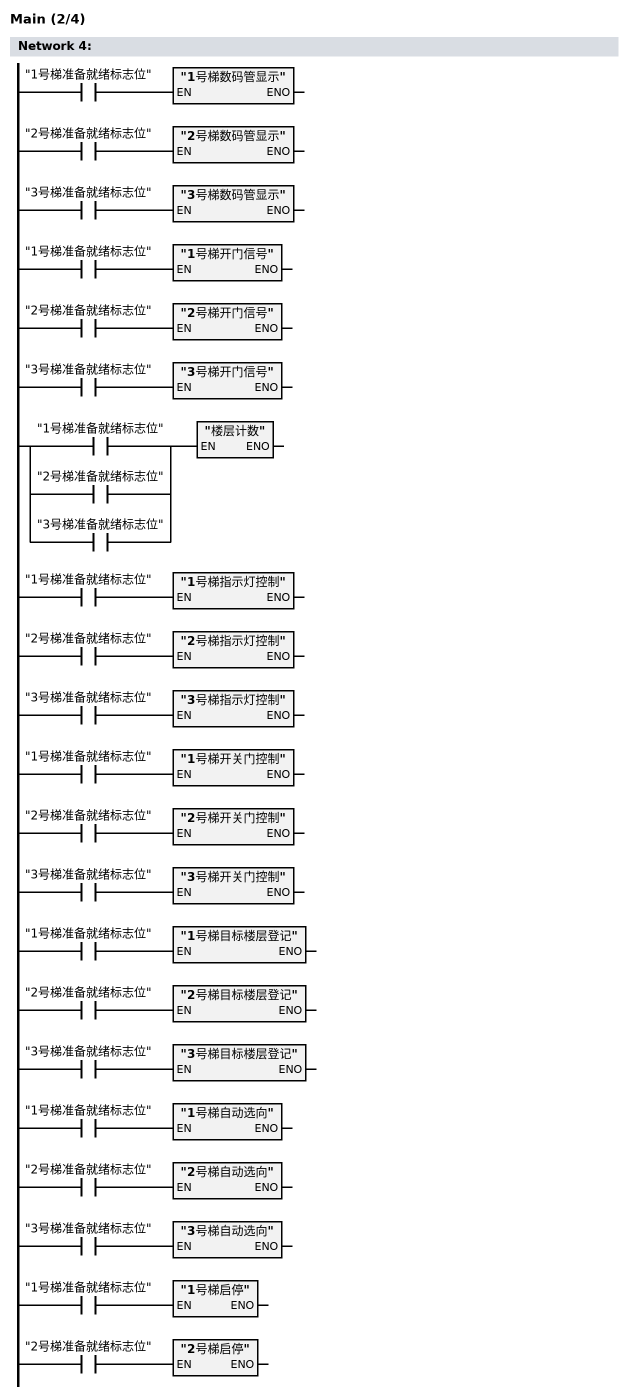
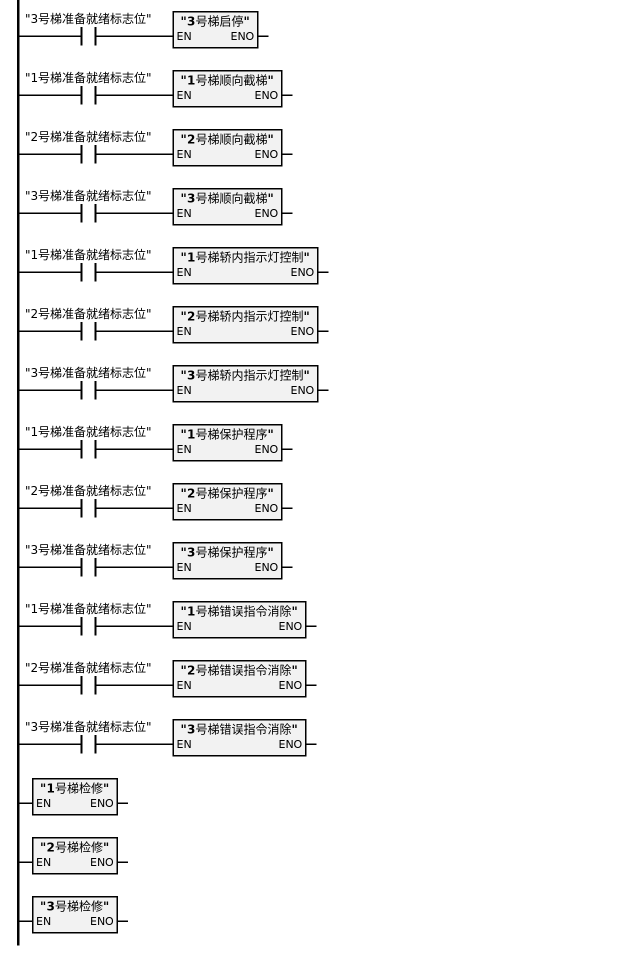
   RUNG wire#powerrail
      Contact( "1号梯准备就绪标志位" )
      "1号梯数码管显示"()
   END_RUNG
   RUNG wire#powerrail
      Contact( "2号梯准备就绪标志位" )
      "2号梯数码管显示"()
   END_RUNG
   RUNG wire#powerrail
      Contact( "3号梯准备就绪标志位" )
      "3号梯数码管显示"()
   END_RUNG
   RUNG wire#powerrail
      Contact( "1号梯准备就绪标志位" )
      "1号梯开门信号"()
   END_RUNG
   RUNG wire#powerrail
      Contact( "2号梯准备就绪标志位" )
      "2号梯开门信号"()
   END_RUNG
   RUNG wire#powerrail
      Contact( "3号梯准备就绪标志位" )
      "3号梯开门信号"()
   END_RUNG
   RUNG wire#powerrail
      Contact( "1号梯准备就绪标志位" )
      wire#w1
      "楼层计数"()
   END_RUNG
   RUNG wire#powerrail
      Contact( "2号梯准备就绪标志位" )
   END_RUNG wire#w1
   RUNG wire#powerrail
      Contact( "3号梯准备就绪标志位" )
   END_RUNG wire#w1
   RUNG wire#powerrail
      Contact( "1号梯准备就绪标志位" )
      "1号梯指示灯控制"()
   END_RUNG
   RUNG wire#powerrail
      Contact( "2号梯准备就绪标志位" )
      "2号梯指示灯控制"()
   END_RUNG
   RUNG wire#powerrail
      Contact( "3号梯准备就绪标志位" )
      "3号梯指示灯控制"()
   END_RUNG
   RUNG wire#powerrail
      Contact( "1号梯准备就绪标志位" )
      "1号梯开关门控制"()
   END_RUNG
   RUNG wire#powerrail
      Contact( "2号梯准备就绪标志位" )
      "2号梯开关门控制"()
   END_RUNG
   RUNG wire#powerrail
      Contact( "3号梯准备就绪标志位" )
      "3号梯开关门控制"()
   END_RUNG
   RUNG wire#powerrail
      Contact( "1号梯准备就绪标志位" )
      "1号梯目标楼层登记"()
   END_RUNG
   RUNG wire#powerrail
      Contact( "2号梯准备就绪标志位" )
      "2号梯目标楼层登记"()
   END_RUNG
   RUNG wire#powerrail
      Contact( "3号梯准备就绪标志位" )
      "3号梯目标楼层登记"()
   END_RUNG
   RUNG wire#powerrail
      Contact( "1号梯准备就绪标志位" )
      "1号梯自动选向"()
   END_RUNG
   RUNG wire#powerrail
      Contact( "2号梯准备就绪标志位" )
      "2号梯自动选向"()
   END_RUNG
   RUNG wire#powerrail
      Contact( "3号梯准备就绪标志位" )
      "3号梯自动选向"()
   END_RUNG
   RUNG wire#powerrail
      Contact( "1号梯准备就绪标志位" )
      "1号梯启停"()
   END_RUNG
   RUNG wire#powerrail
      Contact( "2号梯准备就绪标志位" )
      "2号梯启停"()
   END_RUNG
   RUNG wire#powerrail
      Contact( "3号梯准备就绪标志位" )
      "3号梯启停"()
   END_RUNG
   RUNG wire#powerrail
      Contact( "1号梯准备就绪标志位" )
      "1号梯顺向截梯"()
   END_RUNG
   RUNG wire#powerrail
      Contact( "2号梯准备就绪标志位" )
      "2号梯顺向截梯"()
   END_RUNG
   RUNG wire#powerrail
      Contact( "3号梯准备就绪标志位" )
      "3号梯顺向截梯"()
   END_RUNG
   RUNG wire#powerrail
      Contact( "1号梯准备就绪标志位" )
      "1号梯轿内指示灯控制"()
   END_RUNG
   RUNG wire#powerrail
      Contact( "2号梯准备就绪标志位" )
      "2号梯轿内指示灯控制"()
   END_RUNG
   RUNG wire#powerrail
      Contact( "3号梯准备就绪标志位" )
      "3号梯轿内指示灯控制"()
   END_RUNG
   RUNG wire#powerrail
      Contact( "1号梯准备就绪标志位" )
      "1号梯保护程序"()
   END_RUNG
   RUNG wire#powerrail
      Contact( "2号梯准备就绪标志位" )
      "2号梯保护程序"()
   END_RUNG
   RUNG wire#powerrail
      Contact( "3号梯准备就绪标志位" )
      "3号梯保护程序"()
   END_RUNG
   RUNG wire#powerrail
      Contact( "1号梯准备就绪标志位" )
      "1号梯错误指令消除"()
   END_RUNG
   RUNG wire#powerrail
      Contact( "2号梯准备就绪标志位" )
      "2号梯错误指令消除"()
   END_RUNG
   RUNG wire#powerrail
      Contact( "3号梯准备就绪标志位" )
      "3号梯错误指令消除"()
   END_RUNG
   RUNG wire#powerrail
      "1号梯检修"()
   END_RUNG
   RUNG wire#powerrail
      "2号梯检修"()
   END_RUNG
   RUNG wire#powerrail
      "3号梯检修"()
   END_RUNG
   // the same network as SCL:
   IF "1号梯准备就绪标志位" THEN "1号梯数码管显示"(); END_IF;
   IF "2号梯准备就绪标志位" THEN "2号梯数码管显示"(); END_IF;
   IF "3号梯准备就绪标志位" THEN "3号梯数码管显示"(); END_IF;
   IF "1号梯准备就绪标志位" THEN "1号梯开门信号"(); END_IF;
   IF "2号梯准备就绪标志位" THEN "2号梯开门信号"(); END_IF;
   IF "3号梯准备就绪标志位" THEN "3号梯开门信号"(); END_IF;
   IF "1号梯准备就绪标志位" OR "2号梯准备就绪标志位" OR "3号梯准备就绪标志位" THEN "楼层计数"(); END_IF;
   IF "1号梯准备就绪标志位" THEN "1号梯指示灯控制"(); END_IF;
   IF "2号梯准备就绪标志位" THEN "2号梯指示灯控制"(); END_IF;
   IF "3号梯准备就绪标志位" THEN "3号梯指示灯控制"(); END_IF;
   IF "1号梯准备就绪标志位" THEN "1号梯开关门控制"(); END_IF;
   IF "2号梯准备就绪标志位" THEN "2号梯开关门控制"(); END_IF;
   IF "3号梯准备就绪标志位" THEN "3号梯开关门控制"(); END_IF;
   IF "1号梯准备就绪标志位" THEN "1号梯目标楼层登记"(); END_IF;
   IF "2号梯准备就绪标志位" THEN "2号梯目标楼层登记"(); END_IF;
   IF "3号梯准备就绪标志位" THEN "3号梯目标楼层登记"(); END_IF;
   IF "1号梯准备就绪标志位" THEN "1号梯自动选向"(); END_IF;
   IF "2号梯准备就绪标志位" THEN "2号梯自动选向"(); END_IF;
   IF "3号梯准备就绪标志位" THEN "3号梯自动选向"(); END_IF;
   IF "1号梯准备就绪标志位" THEN "1号梯启停"(); END_IF;
   IF "2号梯准备就绪标志位" THEN "2号梯启停"(); END_IF;
   IF "3号梯准备就绪标志位" THEN "3号梯启停"(); END_IF;
   IF "1号梯准备就绪标志位" THEN "1号梯顺向截梯"(); END_IF;
   IF "2号梯准备就绪标志位" THEN "2号梯顺向截梯"(); END_IF;
   IF "3号梯准备就绪标志位" THEN "3号梯顺向截梯"(); END_IF;
   IF "1号梯准备就绪标志位" THEN "1号梯轿内指示灯控制"(); END_IF;
   IF "2号梯准备就绪标志位" THEN "2号梯轿内指示灯控制"(); END_IF;
   IF "3号梯准备就绪标志位" THEN "3号梯轿内指示灯控制"(); END_IF;
   IF "1号梯准备就绪标志位" THEN "1号梯保护程序"(); END_IF;
   IF "2号梯准备就绪标志位" THEN "2号梯保护程序"(); END_IF;
   IF "3号梯准备就绪标志位" THEN "3号梯保护程序"(); END_IF;
   IF "1号梯准备就绪标志位" THEN "1号梯错误指令消除"(); END_IF;
   IF "2号梯准备就绪标志位" THEN "2号梯错误指令消除"(); END_IF;
   IF "3号梯准备就绪标志位" THEN "3号梯错误指令消除"(); END_IF;
   "1号梯检修"();
   "2号梯检修"();
   "3号梯检修"();
END_REGION

REGION Network 5: 群控
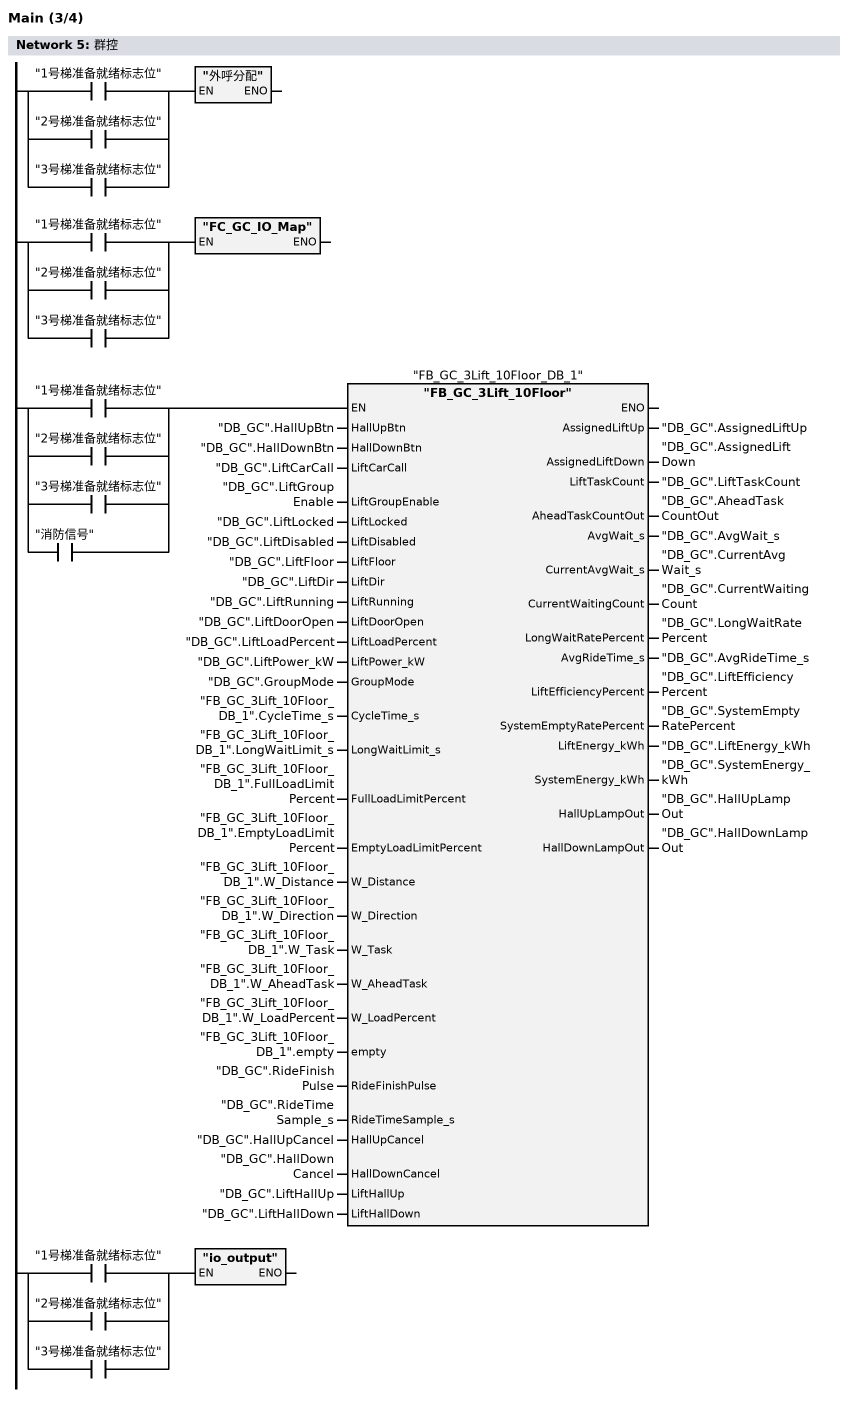
   RUNG wire#powerrail
      Contact( "1号梯准备就绪标志位" )
      wire#w1
      "外呼分配"()
   END_RUNG
   RUNG wire#powerrail
      Contact( "2号梯准备就绪标志位" )
   END_RUNG wire#w1
   RUNG wire#powerrail
      Contact( "3号梯准备就绪标志位" )
   END_RUNG wire#w1
   RUNG wire#powerrail
      Contact( "1号梯准备就绪标志位" )
      wire#w2
      "FC_GC_IO_Map"()
   END_RUNG
   RUNG wire#powerrail
      Contact( "2号梯准备就绪标志位" )
   END_RUNG wire#w2
   RUNG wire#powerrail
      Contact( "3号梯准备就绪标志位" )
   END_RUNG wire#w2
   RUNG wire#powerrail
      Contact( "1号梯准备就绪标志位" )
      wire#w3
      "FB_GC_3Lift_10Floor_DB_1"(HallUpBtn := "DB_GC".HallUpBtn, HallDownBtn := "DB_GC".HallDownBtn, LiftCarCall := "DB_GC".LiftCarCall, LiftGroupEnable := "DB_GC".LiftGroupEnable, LiftLocked := "DB_GC".LiftLocked, LiftDisabled := "DB_GC".LiftDisabled, LiftFloor := "DB_GC".LiftFloor, LiftDir := "DB_GC".LiftDir, LiftRunning := "DB_GC".LiftRunning, LiftDoorOpen := "DB_GC".LiftDoorOpen, LiftLoadPercent := "DB_GC".LiftLoadPercent, LiftPower_kW := "DB_GC".LiftPower_kW, GroupMode := "DB_GC".GroupMode, CycleTime_s := "FB_GC_3Lift_10Floor_DB_1".CycleTime_s, LongWaitLimit_s := "FB_GC_3Lift_10Floor_DB_1".LongWaitLimit_s, FullLoadLimitPercent := "FB_GC_3Lift_10Floor_DB_1".FullLoadLimitPercent, EmptyLoadLimitPercent := "FB_GC_3Lift_10Floor_DB_1".EmptyLoadLimitPercent, W_Distance := "FB_GC_3Lift_10Floor_DB_1".W_Distance, W_Direction := "FB_GC_3Lift_10Floor_DB_1".W_Direction, W_Task := "FB_GC_3Lift_10Floor_DB_1".W_Task, W_AheadTask := "FB_GC_3Lift_10Floor_DB_1".W_AheadTask, W_LoadPercent := "FB_GC_3Lift_10Floor_DB_1".W_LoadPercent, empty := "FB_GC_3Lift_10Floor_DB_1".empty, RideFinishPulse := "DB_GC".RideFinishPulse, RideTimeSample_s := "DB_GC".RideTimeSample_s, HallUpCancel := "DB_GC".HallUpCancel, HallDownCancel := "DB_GC".HallDownCancel, LiftHallUp := "DB_GC".LiftHallUp, LiftHallDown := "DB_GC".LiftHallDown, AssignedLiftUp => "DB_GC".AssignedLiftUp, AssignedLiftDown => "DB_GC".AssignedLiftDown, LiftTaskCount => "DB_GC".LiftTaskCount, AheadTaskCountOut => "DB_GC".AheadTaskCountOut, AvgWait_s => "DB_GC".AvgWait_s, CurrentAvgWait_s => "DB_GC".CurrentAvgWait_s, CurrentWaitingCount => "DB_GC".CurrentWaitingCount, LongWaitRatePercent => "DB_GC".LongWaitRatePercent, AvgRideTime_s => "DB_GC".AvgRideTime_s, LiftEfficiencyPercent => "DB_GC".LiftEfficiencyPercent, SystemEmptyRatePercent => "DB_GC".SystemEmptyRatePercent, LiftEnergy_kWh => "DB_GC".LiftEnergy_kWh, SystemEnergy_kWh => "DB_GC".SystemEnergy_kWh, HallUpLampOut => "DB_GC".HallUpLampOut, HallDownLampOut => "DB_GC".HallDownLampOut)
   END_RUNG
   RUNG wire#powerrail
      Contact( "2号梯准备就绪标志位" )
   END_RUNG wire#w3
   RUNG wire#powerrail
      Contact( "3号梯准备就绪标志位" )
   END_RUNG wire#w3
   RUNG wire#powerrail
      Contact( "消防信号" )
   END_RUNG wire#w3
   RUNG wire#powerrail
      Contact( "1号梯准备就绪标志位" )
      wire#w4
      "io_output"()
   END_RUNG
   RUNG wire#powerrail
      Contact( "2号梯准备就绪标志位" )
   END_RUNG wire#w4
   RUNG wire#powerrail
      Contact( "3号梯准备就绪标志位" )
   END_RUNG wire#w4
   // the same network as SCL:
   IF "1号梯准备就绪标志位" OR "2号梯准备就绪标志位" OR "3号梯准备就绪标志位" THEN "外呼分配"(); END_IF;
   IF "1号梯准备就绪标志位" OR "2号梯准备就绪标志位" OR "3号梯准备就绪标志位" THEN "FC_GC_IO_Map"(); END_IF;
   IF "1号梯准备就绪标志位" OR "2号梯准备就绪标志位" OR "3号梯准备就绪标志位" OR "消防信号" THEN
       "FB_GC_3Lift_10Floor_DB_1"(HallUpBtn := "DB_GC".HallUpBtn,   // "FB_GC_3Lift_10Floor"
                               HallDownBtn := "DB_GC".HallDownBtn,
                               LiftCarCall := "DB_GC".LiftCarCall,
                               LiftGroupEnable := "DB_GC".LiftGroupEnable,
                               LiftLocked := "DB_GC".LiftLocked,
                               LiftDisabled := "DB_GC".LiftDisabled,
                               LiftFloor := "DB_GC".LiftFloor,
                               LiftDir := "DB_GC".LiftDir,
                               LiftRunning := "DB_GC".LiftRunning,
                               LiftDoorOpen := "DB_GC".LiftDoorOpen,
                               LiftLoadPercent := "DB_GC".LiftLoadPercent,
                               LiftPower_kW := "DB_GC".LiftPower_kW,
                               GroupMode := "DB_GC".GroupMode,
                               CycleTime_s := "FB_GC_3Lift_10Floor_DB_1".CycleTime_s,
                               LongWaitLimit_s := "FB_GC_3Lift_10Floor_DB_1".LongWaitLimit_s,
                               FullLoadLimitPercent := "FB_GC_3Lift_10Floor_DB_1".FullLoadLimitPercent,
                               EmptyLoadLimitPercent := "FB_GC_3Lift_10Floor_DB_1".EmptyLoadLimitPercent,
                               W_Distance := "FB_GC_3Lift_10Floor_DB_1".W_Distance,
                               W_Direction := "FB_GC_3Lift_10Floor_DB_1".W_Direction,
                               W_Task := "FB_GC_3Lift_10Floor_DB_1".W_Task,
                               W_AheadTask := "FB_GC_3Lift_10Floor_DB_1".W_AheadTask,
                               W_LoadPercent := "FB_GC_3Lift_10Floor_DB_1".W_LoadPercent,
                               empty := "FB_GC_3Lift_10Floor_DB_1".empty,
                               RideFinishPulse := "DB_GC".RideFinishPulse,
                               RideTimeSample_s := "DB_GC".RideTimeSample_s,
                               HallUpCancel := "DB_GC".HallUpCancel,
                               HallDownCancel := "DB_GC".HallDownCancel,
                               LiftHallUp := "DB_GC".LiftHallUp,
                               LiftHallDown := "DB_GC".LiftHallDown,
                               AssignedLiftUp => "DB_GC".AssignedLiftUp,
                               AssignedLiftDown => "DB_GC".AssignedLiftDown,
                               LiftTaskCount => "DB_GC".LiftTaskCount,
                               AheadTaskCountOut => "DB_GC".AheadTaskCountOut,
                               AvgWait_s => "DB_GC".AvgWait_s,
                               CurrentAvgWait_s => "DB_GC".CurrentAvgWait_s,
                               CurrentWaitingCount => "DB_GC".CurrentWaitingCount,
                               LongWaitRatePercent => "DB_GC".LongWaitRatePercent,
                               AvgRideTime_s => "DB_GC".AvgRideTime_s,
                               LiftEfficiencyPercent => "DB_GC".LiftEfficiencyPercent,
                               SystemEmptyRatePercent => "DB_GC".SystemEmptyRatePercent,
                               LiftEnergy_kWh => "DB_GC".LiftEnergy_kWh,
                               SystemEnergy_kWh => "DB_GC".SystemEnergy_kWh,
                               HallUpLampOut => "DB_GC".HallUpLampOut,
                               HallDownLampOut => "DB_GC".HallDownLampOut);
   END_IF;
   IF "1号梯准备就绪标志位" OR "2号梯准备就绪标志位" OR "3号梯准备就绪标志位" THEN "io_output"(); END_IF;
END_REGION

REGION Network 6: 消防模式
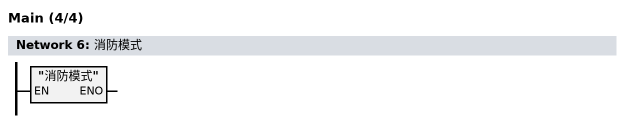
   RUNG wire#powerrail
      "消防模式"()
   END_RUNG
   // the same network as SCL:
   "消防模式"();
END_REGION
END_ORGANIZATION_BLOCK

(* ===== HMI "HMI_RT_1" =====
system functions are stored by id; their names below are inferred from use
connection "HMI_连接_1": ETHERNET, S7_1200_OMS

HMI tags "默认变量表"
   "密码" : WString[254], internal
   "output_准备就绪信号" : Bool = PLC output.准备就绪信号 AT %DB11.DBX17.2, 100 ms
   "input_自动运行信号" : Bool = PLC input.自动运行信号 AT %DB10.DBX14.5, 100 ms
   "output_1号梯故障指示" : Bool = PLC output.1号梯故障指示 AT %DB11.DBX5.4, 100 ms
   "output_1号梯满载指示" : Bool = PLC output.1号梯满载指示 AT %DB11.DBX5.7, 100 ms
   "output_1号梯风扇指示" : Bool = PLC output.1号梯风扇指示 AT %DB11.DBX5.6, 100 ms
   "output_1号梯照明指示" : Bool = PLC output.1号梯照明指示 AT %DB11.DBX5.5, 100 ms
   "当前楼层数" : Int = PLC 1号梯当前楼层数 AT %MW2000, 100 ms
   "上行指示" : Bool = PLC 1号梯上行指示 AT %M23.4, 100 ms
   "下行指示" : Bool = PLC 1号梯下行指示 AT %M2.5, 100 ms
   "output_1号梯开门继电器" : Bool = PLC output.1号梯开门继电器 AT %DB11.DBX6.5, 1 s
   "output_1号梯关门继电器" : Bool = PLC output.1号梯关门继电器 AT %DB11.DBX6.6, 1 s
   "1号梯超重信号" : Bool = PLC 1号梯超重信号 AT %M16.0, 1 s
   "1号梯故障指示" : Bool = PLC 1号梯故障指示 AT %M23.5, 1 s
   "output_1号梯上行指示" : Bool = PLC output.1号梯上行指示 AT %DB11.DBX5.2, 1 s
   "output_1号梯下行指示" : Bool = PLC output.1号梯下行指示 AT %DB11.DBX5.3, 1 s
   "消防信号" : Bool = PLC 消防信号 AT %M1200.0, 1 s
   "2号梯当前楼层数" : Int = PLC 2号梯当前楼层数 AT %MW2100, 1 s
   "3号梯当前楼层数" : Int = PLC 3号梯当前楼层数 AT %MW2300, 1 s
   "1号梯独立运行模式" : Bool = PLC 1号梯独立运行模式 AT %M1201.1, 1 s
   "2号梯独立运行模式" : Bool = PLC 2号梯独立运行模式 AT %M1201.2, 1 s
   "3号梯独立运行模式" : Bool = PLC 3号梯独立运行模式 AT %M1201.3, 1 s
   "output_2号梯上行指示" : Bool = PLC output.2号梯上行指示 AT %DB11.DBX10.2, 1 s
   "output_2号梯下行指示" : Bool = PLC output.2号梯下行指示 AT %DB11.DBX10.3, 1 s
   "output_3号梯上行指示" : Bool = PLC output.3号梯上行指示 AT %DB11.DBX15.2, 1 s
   "output_3号梯下行指示" : Bool = PLC output.3号梯下行指示 AT %DB11.DBX15.3, 1 s
   "output_2号梯故障指示" : Bool = PLC output.2号梯故障指示 AT %DB11.DBX10.4, 1 s
   "output_3号梯故障指示" : Bool = PLC output.3号梯故障指示 AT %DB11.DBX15.4, 1 s
   "output_3号梯照明指示" : Bool = PLC output.3号梯照明指示 AT %DB11.DBX15.5, 1 s
   "output_3号梯风扇指示" : Bool = PLC output.3号梯风扇指示 AT %DB11.DBX15.6, 1 s
   "output_2号梯照明指示" : Bool = PLC output.2号梯照明指示 AT %DB11.DBX10.5, 1 s
   "output_2号梯风扇指示" : Bool = PLC output.2号梯风扇指示 AT %DB11.DBX10.6, 1 s
   "2号梯超重信号" : Bool = PLC 2号梯超重信号 AT %M9.5, 1 s
   "3号梯超重信号" : Bool = PLC 3号梯超重信号 AT %M30.2, 1 s
   "第二次自动运行信号" : Bool = PLC 第二次自动运行信号 AT %M1201.4, 1 s
   "向上初始化使能" : Bool = PLC 向上初始化使能 AT %M1201.5, 1 s

HMI tags "外呼内呼"
   "output_1层上行呼梯按钮指示灯" : Bool = PLC output.1层上行呼梯按钮指示灯 AT %DB11.DBX0.0, 1 s
   "output_2层上行呼梯按钮指示灯" : Bool = PLC output.2层上行呼梯按钮指示灯 AT %DB11.DBX0.1, 1 s
   "output_3层上行呼梯按钮指示灯" : Bool = PLC output.3层上行呼梯按钮指示灯 AT %DB11.DBX0.2, 1 s
   "output_4层上行呼梯按钮指示灯" : Bool = PLC output.4层上行呼梯按钮指示灯 AT %DB11.DBX0.3, 1 s
   "output_5层上行呼梯按钮指示灯" : Bool = PLC output.5层上行呼梯按钮指示灯 AT %DB11.DBX0.4, 1 s
   "output_2层下行呼梯按钮指示灯" : Bool = PLC output.2层下行呼梯按钮指示灯 AT %DB11.DBX1.1, 1 s
   "output_3层下行呼梯按钮指示灯" : Bool = PLC output.3层下行呼梯按钮指示灯 AT %DB11.DBX1.2, 1 s
   "output_4层下行呼梯按钮指示灯" : Bool = PLC output.4层下行呼梯按钮指示灯 AT %DB11.DBX1.3, 1 s
   "output_5层下行呼梯按钮指示灯" : Bool = PLC output.5层下行呼梯按钮指示灯 AT %DB11.DBX1.4, 1 s
   "output_6层下行呼梯按钮指示灯" : Bool = PLC output.6层下行呼梯按钮指示灯 AT %DB11.DBX1.5, 1 s
   "output_1号梯1层按钮指示灯" : Bool = PLC output.1号梯1层按钮指示灯 AT %DB11.DBX2.2, 1 s
   "output_1号梯2层按钮指示灯" : Bool = PLC output.1号梯2层按钮指示灯 AT %DB11.DBX2.3, 1 s
   "output_1号梯3层按钮指示灯" : Bool = PLC output.1号梯3层按钮指示灯 AT %DB11.DBX2.4, 1 s
   "output_1号梯4层按钮指示灯" : Bool = PLC output.1号梯4层按钮指示灯 AT %DB11.DBX2.5, 1 s
   "output_1号梯5层按钮指示灯" : Bool = PLC output.1号梯5层按钮指示灯 AT %DB11.DBX2.6, 1 s
   "output_1号梯6层按钮指示灯" : Bool = PLC output.1号梯6层按钮指示灯 AT %DB11.DBX2.7, 1 s
   "output_6层上行呼梯按钮指示灯" : Bool = PLC output.6层上行呼梯按钮指示灯 AT %DB11.DBX0.5, 1 s
   "output_7层上行呼梯按钮指示灯" : Bool = PLC output.7层上行呼梯按钮指示灯 AT %DB11.DBX0.6, 1 s
   "output_7层下行呼梯按钮指示灯" : Bool = PLC output.7层下行呼梯按钮指示灯 AT %DB11.DBX1.6, 1 s
   "output_8层上行呼梯按钮指示灯" : Bool = PLC output.8层上行呼梯按钮指示灯 AT %DB11.DBX0.7, 1 s
   "output_8层下行呼梯按钮指示灯" : Bool = PLC output.8层下行呼梯按钮指示灯 AT %DB11.DBX1.7, 1 s
   "output_9层上行呼梯按钮指示灯" : Bool = PLC output.9层上行呼梯按钮指示灯 AT %DB11.DBX1.0, 1 s
   "output_9层下行呼梯按钮指示灯" : Bool = PLC output.9层下行呼梯按钮指示灯 AT %DB11.DBX2.0, 1 s
   "output_1号梯7层按钮指示灯" : Bool = PLC output.1号梯7层按钮指示灯 AT %DB11.DBX3.0, 1 s
   "output_1号梯8层按钮指示灯" : Bool = PLC output.1号梯8层按钮指示灯 AT %DB11.DBX3.1, 1 s
   "output_1号梯9层按钮指示灯" : Bool = PLC output.1号梯9层按钮指示灯 AT %DB11.DBX3.2, 1 s
   "output_1号梯10层按钮指示灯" : Bool = PLC output.1号梯10层按钮指示灯 AT %DB11.DBX3.3, 1 s
   "output_10层下行呼梯按钮指示灯" : Bool = PLC output.10层下行呼梯按钮指示灯 AT %DB11.DBX2.1, 1 s
   "output_2号梯1层按钮指示灯" : Bool = PLC output.2号梯1层按钮指示灯 AT %DB11.DBX7.2, 1 s
   "output_2号梯2层按钮指示灯" : Bool = PLC output.2号梯2层按钮指示灯 AT %DB11.DBX7.3, 1 s
   "output_2号梯3层按钮指示灯" : Bool = PLC output.2号梯3层按钮指示灯 AT %DB11.DBX7.4, 1 s
   "output_2号梯4层按钮指示灯" : Bool = PLC output.2号梯4层按钮指示灯 AT %DB11.DBX7.5, 1 s
   "output_2号梯5层按钮指示灯" : Bool = PLC output.2号梯5层按钮指示灯 AT %DB11.DBX7.6, 1 s
   "output_2号梯6层按钮指示灯" : Bool = PLC output.2号梯6层按钮指示灯 AT %DB11.DBX7.7, 1 s
   "output_2号梯7层按钮指示灯" : Bool = PLC output.2号梯7层按钮指示灯 AT %DB11.DBX8.0, 1 s
   "output_2号梯8层按钮指示灯" : Bool = PLC output.2号梯8层按钮指示灯 AT %DB11.DBX8.1, 1 s
   "output_2号梯9层按钮指示灯" : Bool = PLC output.2号梯9层按钮指示灯 AT %DB11.DBX8.2, 1 s
   "output_2号梯10层按钮指示灯" : Bool = PLC output.2号梯10层按钮指示灯 AT %DB11.DBX8.3, 1 s
   "output_3号梯1层按钮指示灯" : Bool = PLC output.3号梯1层按钮指示灯 AT %DB11.DBX12.2, 1 s
   "output_3号梯2层按钮指示灯" : Bool = PLC output.3号梯2层按钮指示灯 AT %DB11.DBX12.3, 1 s
   "output_3号梯3层按钮指示灯" : Bool = PLC output.3号梯3层按钮指示灯 AT %DB11.DBX12.4, 1 s
   "output_3号梯4层按钮指示灯" : Bool = PLC output.3号梯4层按钮指示灯 AT %DB11.DBX12.5, 1 s
   "output_3号梯5层按钮指示灯" : Bool = PLC output.3号梯5层按钮指示灯 AT %DB11.DBX12.6, 1 s
   "output_3号梯6层按钮指示灯" : Bool = PLC output.3号梯6层按钮指示灯 AT %DB11.DBX12.7, 1 s
   "output_3号梯7层按钮指示灯" : Bool = PLC output.3号梯7层按钮指示灯 AT %DB11.DBX13.0, 1 s
   "output_3号梯8层按钮指示灯" : Bool = PLC output.3号梯8层按钮指示灯 AT %DB11.DBX13.1, 1 s
   "output_3号梯9层按钮指示灯" : Bool = PLC output.3号梯9层按钮指示灯 AT %DB11.DBX13.2, 1 s
   "output_3号梯10层按钮指示灯" : Bool = PLC output.3号梯10层按钮指示灯 AT %DB11.DBX13.3, 1 s

HMI tags "数码管"
   "output_1号梯LEDa" : Bool = PLC output.1号梯LEDa AT %DB11.DBX3.4, 1 s
   "output_1号梯LEDb" : Bool = PLC output.1号梯LEDb AT %DB11.DBX3.5, 1 s
   "output_1号梯LEDc" : Bool = PLC output.1号梯LEDc AT %DB11.DBX3.6, 1 s
   "output_1号梯LEDd" : Bool = PLC output.1号梯LEDd AT %DB11.DBX3.7, 1 s
   "output_1号梯LEDe" : Bool = PLC output.1号梯LEDe AT %DB11.DBX4.0, 1 s
   "output_1号梯LEDf" : Bool = PLC output.1号梯LEDf AT %DB11.DBX4.1, 1 s
   "output_1号梯LEDg" : Bool = PLC output.1号梯LEDg AT %DB11.DBX4.2, 1 s
   "output_1号梯LEDh" : Bool = PLC output.1号梯LEDh AT %DB11.DBX4.3, 1 s
   "output_1号梯LEDi" : Bool = PLC output.1号梯LEDi AT %DB11.DBX4.4, 1 s
   "output_1号梯LEDj" : Bool = PLC output.1号梯LEDj AT %DB11.DBX4.5, 1 s
   "output_1号梯LEDk" : Bool = PLC output.1号梯LEDk AT %DB11.DBX4.6, 1 s
   "output_1号梯LEDl" : Bool = PLC output.1号梯LEDl AT %DB11.DBX4.7, 1 s
   "output_1号梯LEDm" : Bool = PLC output.1号梯LEDm AT %DB11.DBX5.0, 1 s
   "output_1号梯LEDn" : Bool = PLC output.1号梯LEDn AT %DB11.DBX5.1, 1 s
   "output_2号梯LEDa" : Bool = PLC output.2号梯LEDa AT %DB11.DBX8.4, 1 s
   "output_2号梯LEDb" : Bool = PLC output.2号梯LEDb AT %DB11.DBX8.5, 1 s
   "output_2号梯LEDc" : Bool = PLC output.2号梯LEDc AT %DB11.DBX8.6, 1 s
   "output_2号梯LEDd" : Bool = PLC output.2号梯LEDd AT %DB11.DBX8.7, 1 s
   "output_2号梯LEDe" : Bool = PLC output.2号梯LEDe AT %DB11.DBX9.0, 1 s
   "output_2号梯LEDf" : Bool = PLC output.2号梯LEDf AT %DB11.DBX9.1, 1 s
   "output_2号梯LEDg" : Bool = PLC output.2号梯LEDg AT %DB11.DBX9.2, 1 s
   "output_2号梯LEDh" : Bool = PLC output.2号梯LEDh AT %DB11.DBX9.3, 1 s
   "output_2号梯LEDi" : Bool = PLC output.2号梯LEDi AT %DB11.DBX9.4, 1 s
   "output_2号梯LEDj" : Bool = PLC output.2号梯LEDj AT %DB11.DBX9.5, 1 s
   "output_2号梯LEDk" : Bool = PLC output.2号梯LEDk AT %DB11.DBX9.6, 1 s
   "output_2号梯LEDl" : Bool = PLC output.2号梯LEDl AT %DB11.DBX9.7, 1 s
   "output_2号梯LEDm" : Bool = PLC output.2号梯LEDm AT %DB11.DBX10.0, 1 s
   "output_2号梯LEDn" : Bool = PLC output.2号梯LEDn AT %DB11.DBX10.1, 1 s
   "output_3号梯LEDa" : Bool = PLC output.3号梯LEDa AT %DB11.DBX13.4, 1 s
   "output_3号梯LEDb" : Bool = PLC output.3号梯LEDb AT %DB11.DBX13.5, 1 s
   "output_3号梯LEDc" : Bool = PLC output.3号梯LEDc AT %DB11.DBX13.6, 1 s
   "output_3号梯LEDd" : Bool = PLC output.3号梯LEDd AT %DB11.DBX13.7, 1 s
   "output_3号梯LEDe" : Bool = PLC output.3号梯LEDe AT %DB11.DBX14.0, 1 s
   "output_3号梯LEDf" : Bool = PLC output.3号梯LEDf AT %DB11.DBX14.1, 1 s
   "output_3号梯LEDg" : Bool = PLC output.3号梯LEDg AT %DB11.DBX14.2, 1 s
   "output_3号梯LEDh" : Bool = PLC output.3号梯LEDh AT %DB11.DBX14.3, 1 s
   "output_3号梯LEDi" : Bool = PLC output.3号梯LEDi AT %DB11.DBX14.4, 1 s
   "output_3号梯LEDj" : Bool = PLC output.3号梯LEDj AT %DB11.DBX14.5, 1 s
   "output_3号梯LEDk" : Bool = PLC output.3号梯LEDk AT %DB11.DBX14.6, 1 s
   "output_3号梯LEDl" : Bool = PLC output.3号梯LEDl AT %DB11.DBX14.7, 1 s
   "output_3号梯LEDm" : Bool = PLC output.3号梯LEDm AT %DB11.DBX15.0, 1 s
   "output_3号梯LEDn" : Bool = PLC output.3号梯LEDn AT %DB11.DBX15.1, 1 s

screen "1号梯电梯显示" 800x600
   TextField "文本域_1" at 97,25 size 34x56; Text '1'
   TextField "文本域_2" at 182,24 size 34x56; Text '2'
   TextField "文本域_3" at 266,24 size 34x56; Text '3'
   Button "按钮_1" at 413,5 size 79x33; TextOff '1号梯'
      on Press: ActivateScreen("1号梯电梯显示", 0)
   Button "按钮_2" at 522,5 size 79x33; TextOff '2号梯'
      on Press: ActivateScreen("2号梯电梯显示", 0)
   Button "按钮_3" at 632,6 size 79x33; TextOff '3号梯'
      on Press: ActivateScreen("3号梯电梯显示", 0)
   TextField "文本域_4" at 429,51 size 57x16; Text '满载指示'
   TextField "文本域_5" at 404,112 size 57x16; Text '运行方向'
   Rectangle "矩形_34" at 559,61 size 35x9
      Appearance <- "output_1号梯LEDa"
   Rectangle "矩形_35" at 560,101 size 35x9
      Appearance <- "output_1号梯LEDg"
   Rectangle "矩形_36" at 560,145 size 35x9
      Appearance <- "output_1号梯LEDd"
   Rectangle "矩形_38" at 593,69 size 9x35
      Appearance <- "output_1号梯LEDb"
   Rectangle "矩形_39" at 551,69 size 9x35
      Appearance <- "output_1号梯LEDf"
   Rectangle "矩形_40" at 594,110 size 9x35
      Appearance <- "output_1号梯LEDc"
   Rectangle "矩形_41" at 552,110 size 9x35
      Appearance <- "output_1号梯LEDe"
   Rectangle "矩形_42" at 504,61 size 35x9
      Appearance <- "output_1号梯LEDh"
   Rectangle "矩形_43" at 504,103 size 35x9
      Appearance <- "output_1号梯LEDn"
   Rectangle "矩形_44" at 504,145 size 35x9
      Appearance <- "output_1号梯LEDk"
   Rectangle "矩形_45" at 538,69 size 9x35
      Appearance <- "output_1号梯LEDi"
   Rectangle "矩形_46" at 496,69 size 9x35
      Appearance <- "output_1号梯LEDm"
   Rectangle "矩形_47" at 538,111 size 9x35
      Appearance <- "output_1号梯LEDj"
   Rectangle "矩形_48" at 496,112 size 9x35
      Appearance <- "output_1号梯LEDl"
   TextField "文本域_6" at 610,55 size 53x15; Text '轿内照明'
   TextField "文本域_7" at 610,100 size 53x15; Text '轿内风扇'
   TextField "文本域_8" at 610,146 size 53x15; Text '故障指示'
   Circle "圆_2" at 666,47 size 34x34
      Appearance <- "output_1号梯照明指示"
   Circle "圆_3" at 666,90 size 34x34
      Appearance <- "output_1号梯风扇指示"
   Circle "圆_4" at 666,133 size 34x34
      Appearance <- "output_1号梯故障指示"
   Circle "圆_1" at 441,67 size 34x34
      Appearance <- "1号梯超重信号"
   TextField "文本域_9" at 447,189 size 27x17; Text '2层'
   TextField "文本域_10" at 479,189 size 27x17; Text '3层'
   TextField "文本域_11" at 512,189 size 27x17; Text '4层'
   TextField "文本域_12" at 544,189 size 27x17; Text '5层'
   TextField "文本域_13" at 576,189 size 27x17; Text '6层'
   TextField "文本域_14" at 609,189 size 27x17; Text '7层'
   TextField "文本域_15" at 641,189 size 27x17; Text '8层'
   TextField "文本域_16" at 673,189 size 27x17; Text '9层'
   TextField "文本域_17" at 705,189 size 35x17; Text '10层'
   TextField "文本域_18" at 415,189 size 27x17; Text '1层'
   Button "按钮_7" at 439,297 size 32x30; TextOff '1'
      Appearance <- "output_1号梯1层按钮指示灯"
   Button "按钮_8" at 485,297 size 32x30; TextOff '2'
      Appearance <- "output_1号梯2层按钮指示灯"
   Button "按钮_9" at 529,297 size 32x30; TextOff '3'
      Appearance <- "output_1号梯3层按钮指示灯"
   Button "按钮_10" at 576,297 size 32x30; TextOff '4'
      Appearance <- "output_1号梯4层按钮指示灯"
   Button "按钮_11" at 623,297 size 32x30; TextOff '5'
      Appearance <- "output_1号梯5层按钮指示灯"
   Button "按钮_12" at 670,297 size 32x30; TextOff '6'
      Appearance <- "output_1号梯6层按钮指示灯"
   Button "按钮_13" at 439,342 size 32x30; TextOff '7'
      Appearance <- "output_1号梯7层按钮指示灯"
   Button "按钮_14" at 483,342 size 32x30; TextOff '8'
      Appearance <- "output_1号梯8层按钮指示灯"
   Button "按钮_15" at 529,342 size 32x30; TextOff '9'
      Appearance <- "output_1号梯9层按钮指示灯"
   Button "按钮_16" at 576,342 size 32x30; TextOff '10'
      Appearance <- "output_1号梯10层按钮指示灯"
   GraphicView "图形视图_18" at 626,347 size 15x23; Picture "Left_Arrow"
   GraphicView "图形视图_20" at 687,347 size 15x23; Picture "Left_Arrow"
   GraphicView "图形视图_21" at 639,347 size 15x23; Picture "Right_Arrow"
   GraphicView "图形视图_22" at 675,347 size 15x23; Picture "Right_Arrow"
   Button "按钮_4" at 626,423 size 72x33; TextOff '消防模式'
      on Press: InvertBit("消防信号")
   TextField "文本域_19" at 446,426 size 103x21; Text '独立运行模式'
   Button "按钮_5" at 434,462 size 44x27; TextOff '1号梯'
      on Press: InvertBit("1号梯独立运行模式")
   Button "按钮_6" at 477,462 size 44x27; TextOff '2号梯'
      on Press: InvertBit("2号梯独立运行模式")
   Button "按钮_17" at 520,462 size 44x27; TextOff '3号梯'
      on Click: InvertBit("3号梯独立运行模式")
   Circle "圆_8" at 638,478 size 45x45
      Appearance <- "消防信号"
   Polygon "多边形_1" at 423,232 size 11x14
      Appearance <- "output_1层上行呼梯按钮指示灯"
   Polygon "多边形_3" at 684,219 size 11x14
      Appearance <- "output_9层上行呼梯按钮指示灯"
   Polygon "多边形_4" at 555,219 size 11x14
      Appearance <- "output_5层上行呼梯按钮指示灯"
   Polygon "多边形_5" at 454,219 size 11x14
      Appearance <- "output_2层上行呼梯按钮指示灯"
   Polygon "多边形_6" at 487,219 size 11x14
      Appearance <- "output_3层上行呼梯按钮指示灯"
   Polygon "多边形_7" at 520,219 size 11x14
      Appearance <- "output_4层上行呼梯按钮指示灯"
   Polygon "多边形_8" at 587,219 size 11x14
      Appearance <- "output_6层上行呼梯按钮指示灯"
   Polygon "多边形_9" at 654,219 size 11x14
      Appearance <- "output_8层上行呼梯按钮指示灯"
   Polygon "多边形_10" at 620,219 size 11x14
      Appearance <- "output_7层上行呼梯按钮指示灯"
   Polygon "多边形_12" at 487,246 size 11x16
      Appearance <- "output_3层下行呼梯按钮指示灯"
   Polygon "多边形_13" at 555,246 size 11x16
      Appearance <- "output_5层下行呼梯按钮指示灯"
   Polygon "多边形_14" at 587,246 size 11x16
      Appearance <- "output_6层下行呼梯按钮指示灯"
   Polygon "多边形_15" at 620,246 size 11x16
      Appearance <- "output_7层下行呼梯按钮指示灯"
   Polygon "多边形_16" at 520,246 size 11x16
      Appearance <- "output_4层下行呼梯按钮指示灯"
   Polygon "多边形_17" at 654,246 size 11x16
      Appearance <- "output_8层下行呼梯按钮指示灯"
   Polygon "多边形_19" at 684,246 size 11x16
      Appearance <- "output_9层下行呼梯按钮指示灯"
   Polygon "多边形_18" at 454,246 size 11x15
      Appearance <- "output_2层下行呼梯按钮指示灯"
   Polygon "多边形_20" at 718,230 size 11x16
      Appearance <- "output_10层下行呼梯按钮指示灯"
   TextField "文本域_20" at 402,128 size 21x19; Text '上'
   TextField "文本域_21" at 441,128 size 21x19; Text '下'
   Circle "圆_9" at 400,151 size 27x27
      Appearance <- "output_1号梯上行指示"
   Circle "圆_10" at 439,151 size 27x27
      Appearance <- "output_1号梯下行指示"
   TextField "文本域_22" at 346,121 size 43x173; Text '1号梯监测'
   Rectangle "矩形_4" at 91,511 size 46x46
      VerticalMovement <- "当前楼层数"
   Rectangle "矩形_1" at 175,511 size 46x46
      VerticalMovement <- "2号梯当前楼层数"
   Rectangle "矩形_5" at 260,511 size 46x46
      VerticalMovement <- "3号梯当前楼层数"
   Circle "圆_5" at 440,508 size 27x27
      Appearance <- "1号梯独立运行模式"
   Circle "圆_6" at 484,508 size 27x27
      Appearance <- "2号梯独立运行模式"
   Circle "圆_7" at 529,508 size 27x27
      Appearance <- "3号梯独立运行模式"
   Button "按钮_18" at 614,535 size 96x32; TextOff '复位使能'
      on Press: SetBit("第二次自动运行信号")
   Button "按钮_19" at 451,540 size 96x32; TextOff '向上初始化'
      on Click: SetBit("向上初始化使能")

screen "2号梯电梯显示" 800x600
   TextField "文本域_4" at 429,51 size 57x16; Text '满载指示'
   TextField "文本域_5" at 404,112 size 57x16; Text '运行方向'
   TextField "文本域_6" at 610,55 size 53x15; Text '轿内照明'
   TextField "文本域_7" at 610,100 size 53x15; Text '轿内风扇'
   TextField "文本域_8" at 610,146 size 53x15; Text '故障指示'
   Circle "圆_2" at 666,47 size 34x34
      Appearance <- "output_2号梯照明指示"
   Circle "圆_3" at 666,90 size 34x34
      Appearance <- "output_2号梯风扇指示"
   Circle "圆_4" at 666,133 size 34x34
      Appearance <- "output_2号梯故障指示"
   Circle "圆_1" at 441,67 size 34x34
      Appearance <- "2号梯超重信号"
   TextField "文本域_9" at 447,189 size 27x17; Text '2层'
   TextField "文本域_10" at 479,189 size 27x17; Text '3层'
   TextField "文本域_11" at 512,189 size 27x17; Text '4层'
   TextField "文本域_12" at 544,189 size 27x17; Text '5层'
   TextField "文本域_13" at 576,189 size 27x17; Text '6层'
   TextField "文本域_14" at 609,189 size 27x17; Text '7层'
   TextField "文本域_15" at 641,189 size 27x17; Text '8层'
   TextField "文本域_16" at 673,189 size 27x17; Text '9层'
   TextField "文本域_17" at 705,189 size 35x17; Text '10层'
   TextField "文本域_18" at 415,189 size 27x17; Text '1层'
   Button "按钮_7" at 439,297 size 32x30; TextOff '1'
      Appearance <- "output_2号梯1层按钮指示灯"
   Button "按钮_8" at 485,297 size 32x30; TextOff '2'
      Appearance <- "output_2号梯2层按钮指示灯"
   Button "按钮_9" at 529,297 size 32x30; TextOff '3'
      Appearance <- "output_2号梯3层按钮指示灯"
   Button "按钮_10" at 576,297 size 32x30; TextOff '4'
      Appearance <- "output_2号梯4层按钮指示灯"
   Button "按钮_11" at 623,297 size 32x30; TextOff '5'
      Appearance <- "output_2号梯5层按钮指示灯"
   Button "按钮_12" at 670,297 size 32x30; TextOff '6'
      Appearance <- "output_2号梯6层按钮指示灯"
   Button "按钮_13" at 439,342 size 32x30; TextOff '7'
      Appearance <- "output_2号梯7层按钮指示灯"
   Button "按钮_14" at 483,342 size 32x30; TextOff '8'
      Appearance <- "output_2号梯8层按钮指示灯"
   Button "按钮_15" at 529,342 size 32x30; TextOff '9'
      Appearance <- "output_2号梯9层按钮指示灯"
   Button "按钮_16" at 576,342 size 32x30; TextOff '10'
      Appearance <- "output_2号梯10层按钮指示灯"
   GraphicView "图形视图_18" at 626,347 size 15x23; Picture "Left_Arrow"
   GraphicView "图形视图_20" at 687,347 size 15x23; Picture "Left_Arrow"
   GraphicView "图形视图_21" at 639,347 size 15x23; Picture "Right_Arrow"
   GraphicView "图形视图_22" at 675,347 size 15x23; Picture "Right_Arrow"
   Button "按钮_4" at 626,423 size 72x33; TextOff '消防模式'
      on Click: InvertBit("消防信号")
   TextField "文本域_19" at 446,426 size 103x21; Text '独立运行模式'
   Button "按钮_5" at 434,462 size 44x27; TextOff '1号梯'
      on Press: InvertBit("1号梯独立运行模式")
   Button "按钮_6" at 477,462 size 44x27; TextOff '2号梯'
      on Press: InvertBit("2号梯独立运行模式")
   Button "按钮_17" at 520,462 size 44x27; TextOff '3号梯'
      on Press: InvertBit("3号梯独立运行模式")
   Circle "圆_8" at 638,478 size 45x45
      Appearance <- "消防信号"
   TextField "文本域_20" at 402,128 size 21x19; Text '上'
   TextField "文本域_21" at 441,128 size 21x19; Text '下'
   Circle "圆_9" at 400,151 size 27x27
      Appearance <- "output_2号梯上行指示"
   Circle "圆_10" at 439,151 size 27x27
      Appearance <- "output_2号梯下行指示"
   Polygon "多边形_1" at 423,232 size 11x14
      Appearance <- "output_1层上行呼梯按钮指示灯"
   Polygon "多边形_3" at 684,219 size 11x14
      Appearance <- "output_9层上行呼梯按钮指示灯"
   Polygon "多边形_4" at 555,219 size 11x14
      Appearance <- "output_5层上行呼梯按钮指示灯"
   Polygon "多边形_5" at 454,219 size 11x14
      Appearance <- "output_2层上行呼梯按钮指示灯"
   Polygon "多边形_6" at 487,219 size 11x14
      Appearance <- "output_3层上行呼梯按钮指示灯"
   Polygon "多边形_7" at 520,219 size 11x14
      Appearance <- "output_4层上行呼梯按钮指示灯"
   Polygon "多边形_8" at 587,219 size 11x14
      Appearance <- "output_6层上行呼梯按钮指示灯"
   Polygon "多边形_9" at 654,219 size 11x14
      Appearance <- "output_8层上行呼梯按钮指示灯"
   Polygon "多边形_10" at 620,219 size 11x14
      Appearance <- "output_7层上行呼梯按钮指示灯"
   Polygon "多边形_12" at 487,246 size 11x16
      Appearance <- "output_3层下行呼梯按钮指示灯"
   Polygon "多边形_13" at 555,246 size 11x16
      Appearance <- "output_5层下行呼梯按钮指示灯"
   Polygon "多边形_14" at 587,246 size 11x16
      Appearance <- "output_6层下行呼梯按钮指示灯"
   Polygon "多边形_15" at 620,246 size 11x16
      Appearance <- "output_7层下行呼梯按钮指示灯"
   Polygon "多边形_16" at 520,246 size 11x16
      Appearance <- "output_4层下行呼梯按钮指示灯"
   Polygon "多边形_17" at 654,246 size 11x16
      Appearance <- "output_8层下行呼梯按钮指示灯"
   Polygon "多边形_19" at 684,246 size 11x16
      Appearance <- "output_9层下行呼梯按钮指示灯"
   Polygon "多边形_18" at 454,246 size 11x15
      Appearance <- "output_2层下行呼梯按钮指示灯"
   Polygon "多边形_20" at 718,230 size 11x16
      Appearance <- "output_10层下行呼梯按钮指示灯"
   Button "按钮_1" at 413,5 size 79x33; TextOff '1号梯'
      on Press: ActivateScreen("1号梯电梯显示", 0)
   Button "按钮_2" at 522,5 size 79x33; TextOff '2号梯'
      on Press: ActivateScreen("2号梯电梯显示", 0)
   Button "按钮_3" at 632,6 size 79x33; TextOff '3号梯'
      on Press: ActivateScreen("3号梯电梯显示", 0)
   TextField "文本域_22" at 346,121 size 43x173; Text '2号梯监测'
   TextField "文本域_1" at 97,25 size 34x56; Text '1'
   TextField "文本域_2" at 182,24 size 34x56; Text '2'
   TextField "文本域_3" at 266,24 size 34x56; Text '3'
   Rectangle "矩形_34" at 559,61 size 35x9
      Appearance <- "output_2号梯LEDa"
   Rectangle "矩形_35" at 560,101 size 35x9
      Appearance <- "output_2号梯LEDg"
   Rectangle "矩形_36" at 560,145 size 35x9
      Appearance <- "output_2号梯LEDd"
   Rectangle "矩形_38" at 593,69 size 9x35
      Appearance <- "output_2号梯LEDb"
   Rectangle "矩形_39" at 551,69 size 9x35
      Appearance <- "output_2号梯LEDf"
   Rectangle "矩形_40" at 594,110 size 9x35
      Appearance <- "output_2号梯LEDc"
   Rectangle "矩形_41" at 552,110 size 9x35
      Appearance <- "output_2号梯LEDe"
   Rectangle "矩形_42" at 504,61 size 35x9
      Appearance <- "output_2号梯LEDh"
   Rectangle "矩形_43" at 504,103 size 35x9
      Appearance <- "output_2号梯LEDn"
   Rectangle "矩形_44" at 504,145 size 35x9
      Appearance <- "output_2号梯LEDk"
   Rectangle "矩形_45" at 538,69 size 9x35
      Appearance <- "output_2号梯LEDi"
   Rectangle "矩形_46" at 496,69 size 9x35
      Appearance <- "output_2号梯LEDm"
   Rectangle "矩形_47" at 538,111 size 9x35
      Appearance <- "output_2号梯LEDj"
   Rectangle "矩形_48" at 496,112 size 9x35
      Appearance <- "output_2号梯LEDl"
   Circle "圆_5" at 440,508 size 27x27
      Appearance <- "1号梯独立运行模式"
   Circle "圆_6" at 484,508 size 27x27
      Appearance <- "2号梯独立运行模式"
   Circle "圆_7" at 529,508 size 27x27
      Appearance <- "3号梯独立运行模式"
   Rectangle "矩形_4" at 91,511 size 46x46
      VerticalMovement <- "当前楼层数"
   Rectangle "矩形_1" at 175,511 size 46x46
      VerticalMovement <- "2号梯当前楼层数"
   Rectangle "矩形_5" at 260,511 size 46x46
      VerticalMovement <- "3号梯当前楼层数"
   Button "按钮_18" at 614,535 size 96x32; TextOff '复位使能'
      on Press: SetBit("第二次自动运行信号")
   Button "按钮_19" at 451,540 size 96x32; TextOff '向上初始化'
      on Click: SetBit("向上初始化使能")

screen "3号梯电梯显示" 800x600
   TextField "文本域_4" at 429,51 size 57x16; Text '满载指示'
   TextField "文本域_5" at 404,112 size 57x16; Text '运行方向'
   TextField "文本域_6" at 610,55 size 53x15; Text '轿内照明'
   TextField "文本域_7" at 610,100 size 53x15; Text '轿内风扇'
   TextField "文本域_8" at 610,146 size 53x15; Text '故障指示'
   Circle "圆_2" at 666,47 size 34x34
      Appearance <- "output_3号梯照明指示"
   Circle "圆_3" at 666,90 size 34x34
      Appearance <- "output_3号梯风扇指示"
   Circle "圆_4" at 666,133 size 34x34
      Appearance <- "output_3号梯故障指示"
   Circle "圆_1" at 441,67 size 34x34
      Appearance <- "3号梯超重信号"
   TextField "文本域_9" at 447,189 size 27x17; Text '2层'
   TextField "文本域_10" at 479,189 size 27x17; Text '3层'
   TextField "文本域_11" at 512,189 size 27x17; Text '4层'
   TextField "文本域_12" at 544,189 size 27x17; Text '5层'
   TextField "文本域_13" at 576,189 size 27x17; Text '6层'
   TextField "文本域_14" at 609,189 size 27x17; Text '7层'
   TextField "文本域_15" at 641,189 size 27x17; Text '8层'
   TextField "文本域_16" at 673,189 size 27x17; Text '9层'
   TextField "文本域_17" at 705,189 size 35x17; Text '10层'
   TextField "文本域_18" at 415,189 size 27x17; Text '1层'
   Button "按钮_7" at 439,297 size 32x30; TextOff '1'
      Appearance <- "output_3号梯1层按钮指示灯"
   Button "按钮_8" at 485,297 size 32x30; TextOff '2'
      Appearance <- "output_3号梯2层按钮指示灯"
   Button "按钮_9" at 529,297 size 32x30; TextOff '3'
      Appearance <- "output_3号梯3层按钮指示灯"
   Button "按钮_10" at 576,297 size 32x30; TextOff '4'
      Appearance <- "output_3号梯4层按钮指示灯"
   Button "按钮_11" at 623,297 size 32x30; TextOff '5'
      Appearance <- "output_3号梯5层按钮指示灯"
   Button "按钮_12" at 670,297 size 32x30; TextOff '6'
      Appearance <- "output_3号梯6层按钮指示灯"
   Button "按钮_13" at 439,342 size 32x30; TextOff '7'
      Appearance <- "output_3号梯7层按钮指示灯"
   Button "按钮_14" at 483,342 size 32x30; TextOff '8'
      Appearance <- "output_3号梯8层按钮指示灯"
   Button "按钮_15" at 529,342 size 32x30; TextOff '9'
      Appearance <- "output_3号梯9层按钮指示灯"
   Button "按钮_16" at 576,342 size 32x30; TextOff '10'
      Appearance <- "output_3号梯10层按钮指示灯"
   GraphicView "图形视图_18" at 626,347 size 15x23; Picture "Left_Arrow"
   GraphicView "图形视图_20" at 687,347 size 15x23; Picture "Left_Arrow"
   GraphicView "图形视图_21" at 639,347 size 15x23; Picture "Right_Arrow"
   GraphicView "图形视图_22" at 675,347 size 15x23; Picture "Right_Arrow"
   Button "按钮_4" at 626,423 size 72x33; TextOff '消防模式'
      on Click: InvertBit("消防信号")
   TextField "文本域_19" at 446,426 size 103x21; Text '独立运行模式'
   Circle "圆_5" at 440,508 size 27x27
      Appearance <- "1号梯独立运行模式"
   Circle "圆_6" at 484,508 size 27x27
      Appearance <- "2号梯独立运行模式"
   Circle "圆_7" at 529,508 size 27x27
      Appearance <- "3号梯独立运行模式"
   Button "按钮_5" at 434,462 size 44x27; TextOff '1号梯'
      on Press: InvertBit("1号梯独立运行模式")
   Button "按钮_6" at 477,462 size 44x27; TextOff '2号梯'
      on Press: InvertBit("2号梯独立运行模式")
   Button "按钮_17" at 520,462 size 44x27; TextOff '3号梯'
      on Click: InvertBit("3号梯独立运行模式")
   Circle "圆_8" at 638,478 size 45x45
      Appearance <- "消防信号"
   Polygon "多边形_1" at 423,232 size 11x14
      Appearance <- "output_1层上行呼梯按钮指示灯"
   Polygon "多边形_3" at 684,219 size 11x14
      Appearance <- "output_9层上行呼梯按钮指示灯"
   Polygon "多边形_4" at 555,219 size 11x14
      Appearance <- "output_5层上行呼梯按钮指示灯"
   Polygon "多边形_5" at 454,219 size 11x14
      Appearance <- "output_2层上行呼梯按钮指示灯"
   Polygon "多边形_6" at 487,219 size 11x14
      Appearance <- "output_3层上行呼梯按钮指示灯"
   Polygon "多边形_7" at 520,219 size 11x14
      Appearance <- "output_4层上行呼梯按钮指示灯"
   Polygon "多边形_8" at 587,219 size 11x14
      Appearance <- "output_6层上行呼梯按钮指示灯"
   Polygon "多边形_9" at 654,219 size 11x14
      Appearance <- "output_8层上行呼梯按钮指示灯"
   Polygon "多边形_10" at 620,219 size 11x14
      Appearance <- "output_7层上行呼梯按钮指示灯"
   Polygon "多边形_12" at 487,246 size 11x16
      Appearance <- "output_3层下行呼梯按钮指示灯"
   Polygon "多边形_13" at 555,246 size 11x16
      Appearance <- "output_5层下行呼梯按钮指示灯"
   Polygon "多边形_14" at 587,246 size 11x16
      Appearance <- "output_6层下行呼梯按钮指示灯"
   Polygon "多边形_15" at 620,246 size 11x16
      Appearance <- "output_7层下行呼梯按钮指示灯"
   Polygon "多边形_16" at 520,246 size 11x16
      Appearance <- "output_4层下行呼梯按钮指示灯"
   Polygon "多边形_17" at 654,246 size 11x16
      Appearance <- "output_8层下行呼梯按钮指示灯"
   Polygon "多边形_19" at 684,246 size 11x16
      Appearance <- "output_9层下行呼梯按钮指示灯"
   Polygon "多边形_18" at 454,246 size 11x15
      Appearance <- "output_2层下行呼梯按钮指示灯"
   Polygon "多边形_20" at 718,230 size 11x16
      Appearance <- "output_10层下行呼梯按钮指示灯"
   TextField "文本域_20" at 402,128 size 21x19; Text '上'
   TextField "文本域_21" at 441,128 size 21x19; Text '下'
   Circle "圆_9" at 400,151 size 27x27
      Appearance <- "output_3号梯上行指示"
   Circle "圆_10" at 439,151 size 27x27
      Appearance <- "output_3号梯下行指示"
   Button "按钮_1" at 413,5 size 79x33; TextOff '1号梯'
      on Press: ActivateScreen("1号梯电梯显示", 0)
   Button "按钮_2" at 522,5 size 79x33; TextOff '2号梯'
      on Press: ActivateScreen("2号梯电梯显示", 0)
   Button "按钮_3" at 632,6 size 79x33; TextOff '3号梯'
      on Press: ActivateScreen("3号梯电梯显示", 0)
   TextField "文本域_22" at 346,121 size 43x173; Text '3号梯监测'
   TextField "文本域_1" at 97,25 size 34x56; Text '1'
   TextField "文本域_2" at 182,24 size 34x56; Text '2'
   TextField "文本域_3" at 266,24 size 34x56; Text '3'
   Rectangle "矩形_34" at 559,61 size 35x9
      Appearance <- "output_3号梯LEDa"
   Rectangle "矩形_35" at 560,101 size 35x9
      Appearance <- "output_3号梯LEDg"
   Rectangle "矩形_36" at 560,145 size 35x9
      Appearance <- "output_3号梯LEDd"
   Rectangle "矩形_38" at 593,69 size 9x35
      Appearance <- "output_3号梯LEDb"
   Rectangle "矩形_39" at 551,69 size 9x35
      Appearance <- "output_3号梯LEDf"
   Rectangle "矩形_40" at 594,110 size 9x35
      Appearance <- "output_3号梯LEDc"
   Rectangle "矩形_41" at 552,110 size 9x35
      Appearance <- "output_3号梯LEDe"
   Rectangle "矩形_42" at 504,61 size 35x9
      Appearance <- "output_3号梯LEDh"
   Rectangle "矩形_43" at 504,103 size 35x9
      Appearance <- "output_3号梯LEDn"
   Rectangle "矩形_44" at 504,145 size 35x9
      Appearance <- "output_3号梯LEDk"
   Rectangle "矩形_45" at 538,69 size 9x35
      Appearance <- "output_3号梯LEDi"
   Rectangle "矩形_46" at 496,69 size 9x35
      Appearance <- "output_3号梯LEDm"
   Rectangle "矩形_47" at 538,111 size 9x35
      Appearance <- "output_3号梯LEDj"
   Rectangle "矩形_48" at 496,112 size 9x35
      Appearance <- "output_3号梯LEDl"
   Rectangle "矩形_4" at 91,511 size 46x46
      VerticalMovement <- "当前楼层数"
   Rectangle "矩形_1" at 175,511 size 46x46
      VerticalMovement <- "2号梯当前楼层数"
   Rectangle "矩形_5" at 260,511 size 46x46
      VerticalMovement <- "3号梯当前楼层数"
   Button "按钮_18" at 614,535 size 96x32; TextOff '复位使能'
      on Press: SetBit("第二次自动运行信号")
   Button "按钮_19" at 451,540 size 96x32; TextOff '向上初始化'
      on Click: SetBit("向上初始化使能")

screen "登录" 800x600
   GraphicView "图形视图_1" at 0,0 size 799x600; Picture "6ece7c403888456fd3f6ea8c2ca127ef"
   IOField "I/O 域_1" at 485,273 size 224x48; FormatPattern ????????????????????????????????????????????????????????????????????????????????
      ProcessValue <- "密码"
   TextField "文本域_1" at 427,276 size 41x36; Text '密码'
   Button "按钮_1" at 528,361 size 96x32; TextOff '登录'
      on Click: ActivateScreen("1号梯电梯显示", 0)
   TextField "文本域_2" at 515,208 size 129x31; Text '管理员登录'

VB script "login"
   Dim pwd
   pwd = SmartTags("密码")
   
   If pwd = "123" Then
      bec8f1e5-2ab1-45f6-ad91-1d37c469eb91 1号梯电梯显示, 0
   Else
       SmartTags("密码") = ""                     ' 清空 I/O 域
   End If
*)